LIN {X 0,Y 573.221,Z 156.08,A -85,B 0,C 180,E1 -2313.023,E2 -2313.023} C_VEL
LIN {X 0,Y 573.249,Z 156.083,A -85,B 0,C 180,E1 -2315.365,E2 -2315.365} C_VEL
LIN {X 0,Y 573.247,Z 156.077,A -85,B 0,C 180,E1 -2317.663,E2 -2317.663} C_VEL
LIN {X 0,Y 573.25,Z 156.08,A -85,B 0,C 180,E1 -2320.726,E2 -2320.726} C_VEL
LIN {X 0,Y 573.241,Z 156.081,A -85,B 0,C 180,E1 -2323.622,E2 -2323.622} C_VEL
LIN {X 0,Y 573.206,Z 156.082,A -85,B 0,C 180,E1 -2326.529,E2 -2326.529} C_VEL
LIN {X 0,Y 573.275,Z 156.074,A -85,B 0,C 180,E1 -2329.404,E2 -2329.404} C_VEL
LIN {X 0,Y 573.284,Z 156.078,A -85,B 0,C 180,E1 -2332.25,E2 -2332.25} C_VEL
LIN {X 0,Y 573.299,Z 156.071,A -85,B 0,C 180,E1 -2335.077,E2 -2335.077} C_VEL
LIN {X 0,Y 573.269,Z 156.075,A -85,B 0,C 180,E1 -2337.892,E2 -2337.892} C_VEL
LIN {X 0,Y 573.318,Z 156.074,A -85,B 0,C 180,E1 -2340.703,E2 -2340.703} C_VEL
LIN {X 0,Y 573.227,Z 156.079,A -85,B 0,C 180,E1 -2343.515,E2 -2343.515} C_VEL
LIN {X 0,Y 573.286,Z 156.077,A -85,B 0,C 180,E1 -2345.628,E2 -2345.628} C_VEL
LIN {X 0,Y 573.282,Z 156.073,A -85,B 0,C 180,E1 -2348.46,E2 -2348.46} C_VEL
LIN {X 0,Y 573.246,Z 156.078,A -85,B 0,C 180,E1 -2351.313,E2 -2351.313} C_VEL
LIN {X 0,Y 573.259,Z 156.078,A -85,B 0,C 180,E1 -2354.429,E2 -2354.429} C_VEL
LIN {X 0,Y 573.274,Z 156.074,A -85,B 0,C 180,E1 -2357.111,E2 -2357.111} C_VEL
LIN {X 0,Y 573.241,Z 156.077,A -85,B 0,C 180,E1 -2360.077,E2 -2360.077} C_VEL
LIN {X 0,Y 573.209,Z 156.082,A -85,B 0,C 180,E1 -2363.101,E2 -2363.101} C_VEL
LIN {X 0,Y 573.226,Z 156.08,A -85,B 0,C 180,E1 -2364.417,E2 -2364.417} C_VEL
LIN {X 0,Y 572.6,Z 156.16,A -85,B 0,C 180,E1 -2365.004,E2 -2365.004} C_VEL
LIN {X 0,Y 569.761,Z 156.517,A -85,B 0,C 180,E1 -2365.955,E2 -2365.955} C_VEL
LIN {X 0,Y 567.333,Z 156.82,A -85,B 0,C 180,E1 -2366.721,E2 -2366.721} C_VEL
LIN {X 0,Y 566.281,Z 156.947,A -85,B 0,C 180,E1 -2367.313,E2 -2367.313} C_VEL
LIN {X 0,Y 566.193,Z 156.957,A -85,B 0,C 180,E1 -2367.513,E2 -2367.513} C_VEL
LIN {X 0,Y 566.176,Z 156.959,A -85,B 0,C 180,E1 -2370.593,E2 -2370.593} C_VEL
LIN {X 0,Y 566.209,Z 156.955,A -85,B 0,C 180,E1 -2373.103,E2 -2373.103} C_VEL
LIN {X 0,Y 566.173,Z 156.961,A -85,B 0,C 180,E1 -2375.692,E2 -2375.692} C_VEL
LIN {X 0,Y 566.193,Z 156.955,A -85,B 0,C 180,E1 -2378.56,E2 -2378.56} C_VEL
LIN {X 0,Y 566.197,Z 156.96,A -85,B 0,C 180,E1 -2381.138,E2 -2381.138} C_VEL
LIN {X 0,Y 566.187,Z 156.958,A -85,B 0,C 180,E1 -2384.037,E2 -2384.037} C_VEL
LIN {X 0,Y 566.19,Z 156.956,A -85,B 0,C 180,E1 -2387.085,E2 -2387.085} C_VEL
LIN {X 0,Y 566.195,Z 156.958,A -85,B 0,C 180,E1 -2389.803,E2 -2389.803} C_VEL
LIN {X 0,Y 566.131,Z 156.967,A -85,B 0,C 180,E1 -2392.537,E2 -2392.537} C_VEL
LIN {X 0,Y 566.126,Z 159.575,A -85,B 0,C 180,E1 -2394.308,E2 -2394.308} C_VEL
LIN {X 0,Y 566.103,Z 163.804,A -85,B 0,C 180,E1 -2396.892,E2 -2396.892} C_VEL
LIN {X 0,Y 566.069,Z 167.996,A -85,B 0,C 180,E1 -2399.402,E2 -2399.402} C_VEL
LIN {X 0,Y 566.072,Z 172.14,A -85,B 0,C 180,E1 -2401.851,E2 -2401.851} C_VEL
LIN {X 0,Y 566.04,Z 177.644,A -85,B 0,C 180,E1 -2405.031,E2 -2405.031} C_VEL
LIN {X 0,Y 565.949,Z 181.747,A -85,B 0,C 180,E1 -2407.36,E2 -2407.36} C_VEL
LIN {X 0,Y 565.931,Z 187.178,A -85,B 0,C 180,E1 -2410.41,E2 -2410.41} C_VEL
LIN {X 0,Y 565.882,Z 192.758,A -85,B 0,C 180,E1 -2413.403,E2 -2413.403} C_VEL
LIN {X 0,Y 565.839,Z 196.558,A -85,B 0,C 180,E1 -2415.415,E2 -2415.415} C_VEL
LIN {X 0,Y 566.895,Z 204.229,A -85,B 0,C 180,E1 -2415.603,E2 -2415.603} C_VEL
LIN {X 0,Y 566.792,Z 217.644,A -85,B 0,C 180,E1 -2416.008,E2 -2416.008} C_VEL
LIN {X 0,Y 566.595,Z 230.276,A -85,B 0,C 180,E1 -2416.552,E2 -2416.552} C_VEL
LIN {X 0,Y 566.435,Z 241.516,A -85,B 0,C 180,E1 -2417.187,E2 -2417.187} C_VEL
LIN {X 0,Y 566.365,Z 252.951,A -85,B 0,C 180,E1 -2418.004,E2 -2418.004} C_VEL
LIN {X 0,Y 566.217,Z 262.307,A -85,B 0,C 180,E1 -2418.835,E2 -2418.835} C_VEL
LIN {X 0,Y 566.14,Z 271.26,A -85,B 0,C 180,E1 -2419.811,E2 -2419.811} C_VEL
LIN {X 0,Y 566.053,Z 279.323,A -85,B 0,C 180,E1 -2420.892,E2 -2420.892} C_VEL
LIN {X 0,Y 565.991,Z 284.78,A -85,B 0,C 180,E1 -2421.79,E2 -2421.79} C_VEL
LIN {X 0,Y 565.972,Z 290.113,A -85,B 0,C 180,E1 -2422.867,E2 -2422.867} C_VEL
LIN {X 0,Y 565.913,Z 294.264,A -85,B 0,C 180,E1 -2423.941,E2 -2423.941} C_VEL
LIN {X 0,Y 565.858,Z 297.355,A -85,B 0,C 180,E1 -2425.012,E2 -2425.012} C_VEL
LIN {X 0,Y 565.914,Z 298.89,A -85,B 0,C 180,E1 -2425.727,E2 -2425.727} C_VEL
LIN {X 0,Y 565.912,Z 299.981,A -85,B 0,C 180,E1 -2426.44,E2 -2426.44} C_VEL
LIN {X 0,Y 565.839,Z 300.967,A -85,B 0,C 180,E1 -2427.864,E2 -2427.864} C_VEL
LIN {X 0,Y 565.845,Z 300.887,A -85,B 0,C 180,E1 -2428.576,E2 -2428.576} C_VEL
LIN {X 0,Y 565.841,Z 300.384,A -85,B 0,C 180,E1 -2429.288,E2 -2429.288} C_VEL
LIN {X 0,Y 565.843,Z 298.185,A -85,B 0,C 180,E1 -2430.711,E2 -2430.711} C_VEL
LIN {X 0,Y 565.908,Z 295.441,A -85,B 0,C 180,E1 -2431.779,E2 -2431.779} C_VEL
LIN {X 0,Y 565.902,Z 291.689,A -85,B 0,C 180,E1 -2432.847,E2 -2432.847} C_VEL
LIN {X 0,Y 566.003,Z 286.823,A -85,B 0,C 180,E1 -2433.915,E2 -2433.915} C_VEL
LIN {X 0,Y 566.047,Z 280.702,A -85,B 0,C 180,E1 -2434.985,E2 -2434.985} C_VEL
LIN {X 0,Y 566.111,Z 273.096,A -85,B 0,C 180,E1 -2436.056,E2 -2436.056} C_VEL
LIN {X 0,Y 566.191,Z 265.345,A -85,B 0,C 180,E1 -2436.948,E2 -2436.948} C_VEL
LIN {X 0,Y 566.321,Z 254.772,A -85,B 0,C 180,E1 -2437.935,E2 -2437.935} C_VEL
LIN {X 0,Y 566.454,Z 244.034,A -85,B 0,C 180,E1 -2438.741,E2 -2438.741} C_VEL
LIN {X 0,Y 566.563,Z 233.576,A -85,B 0,C 180,E1 -2439.369,E2 -2439.369} C_VEL
LIN {X 0,Y 566.742,Z 221.019,A -85,B 0,C 180,E1 -2439.951,E2 -2439.951} C_VEL
LIN {X 0,Y 566.873,Z 207.708,A -85,B 0,C 180,E1 -2440.4,E2 -2440.4} C_VEL
LIN {X 0,Y 566.719,Z 201.824,A -85,B 0,C 180,E1 -2440.55,E2 -2440.55} C_VEL
LIN {X 0,Y 565.896,Z 196.528,A -85,B 0,C 180,E1 -2440.69,E2 -2440.69} C_VEL
LIN {X 0,Y 565.922,Z 190.956,A -85,B 0,C 180,E1 -2443.646,E2 -2443.646} C_VEL
LIN {X 0,Y 565.91,Z 186.866,A -85,B 0,C 180,E1 -2445.854,E2 -2445.854} C_VEL
LIN {X 0,Y 565.974,Z 182.892,A -85,B 0,C 180,E1 -2448.084,E2 -2448.084} C_VEL
LIN {X 0,Y 566.027,Z 177.535,A -85,B 0,C 180,E1 -2451.103,E2 -2451.103} C_VEL
LIN {X 0,Y 566.052,Z 172.237,A -85,B 0,C 180,E1 -2454.185,E2 -2454.185} C_VEL
LIN {X 0,Y 566.089,Z 166.881,A -85,B 0,C 180,E1 -2457.343,E2 -2457.343} C_VEL
LIN {X 0,Y 566.106,Z 162.848,A -85,B 0,C 180,E1 -2459.771,E2 -2459.771} C_VEL
LIN {X 0,Y 566.117,Z 158.483,A -85,B 0,C 180,E1 -2462.415,E2 -2462.415} C_VEL
LIN {X 0,Y 566.1,Z 157.355,A -85,B 0,C 180,E1 -2463.107,E2 -2463.107} C_VEL
LIN {X 0,Y 566.162,Z 156.96,A -85,B 0,C 180,E1 -2463.956,E2 -2463.956} C_VEL
LIN {X 0,Y 566.168,Z 156.963,A -85,B 0,C 180,E1 -2466.569,E2 -2466.569} C_VEL
LIN {X 0,Y 566.199,Z 156.954,A -85,B 0,C 180,E1 -2469.271,E2 -2469.271} C_VEL
LIN {X 0,Y 566.209,Z 156.958,A -85,B 0,C 180,E1 -2472.083,E2 -2472.083} C_VEL
LIN {X 0,Y 566.154,Z 156.961,A -85,B 0,C 180,E1 -2475.033,E2 -2475.033} C_VEL
LIN {X 0,Y 566.209,Z 156.952,A -85,B 0,C 180,E1 -2478.132,E2 -2478.132} C_VEL
LIN {X 0,Y 566.199,Z 156.961,A -85,B 0,C 180,E1 -2480.725,E2 -2480.725} C_VEL
LIN {X 0,Y 566.175,Z 156.96,A -85,B 0,C 180,E1 -2483.783,E2 -2483.783} C_VEL
LIN {X 0,Y 566.202,Z 156.954,A -85,B 0,C 180,E1 -2486.896,E2 -2486.896} C_VEL
LIN {X 0,Y 566.17,Z 156.964,A -85,B 0,C 180,E1 -2489.406,E2 -2489.406} C_VEL
LIN {X 0,Y 566.196,Z 156.954,A -85,B 0,C 180,E1 -2491.856,E2 -2491.856} C_VEL
LIN {X 0,Y 566.202,Z 156.956,A -85,B 0,C 180,E1 -2494.25,E2 -2494.25} C_VEL
LIN {X 0,Y 566.22,Z 156.954,A -85,B 0,C 180,E1 -2496.697,E2 -2496.697} C_VEL
LIN {X 0,Y 566.184,Z 156.96,A -85,B 0,C 180,E1 -2499.661,E2 -2499.661} C_VEL
LIN {X 0,Y 566.214,Z 156.954,A -85,B 0,C 180,E1 -2502.875,E2 -2502.875} C_VEL
LIN {X 0,Y 566.205,Z 156.955,A -85,B 0,C 180,E1 -2505.626,E2 -2505.626} C_VEL
LIN {X 0,Y 566.254,Z 156.953,A -85,B 0,C 180,E1 -2508.643,E2 -2508.643} C_VEL
LIN {X 0,Y 566.226,Z 156.951,A -85,B 0,C 180,E1 -2511.434,E2 -2511.434} C_VEL
LIN {X 0,Y 566.212,Z 156.956,A -85,B 0,C 180,E1 -2513.586,E2 -2513.586} C_VEL
LIN {X 0,Y 566.165,Z 156.963,A -85,B 0,C 180,E1 -2515.728,E2 -2515.728} C_VEL
LIN {X 0,Y 566.236,Z 156.951,A -85,B 0,C 180,E1 -2517.866,E2 -2517.866} C_VEL
LIN {X 0,Y 566.278,Z 156.95,A -85,B 0,C 180,E1 -2520.711,E2 -2520.711} C_VEL
LIN {X 0,Y 566.17,Z 156.958,A -85,B 0,C 180,E1 -2523.558,E2 -2523.558} C_VEL
LIN {X 0,Y 566.25,Z 156.951,A -85,B 0,C 180,E1 -2525.698,E2 -2525.698} C_VEL
LIN {X 0,Y 566.229,Z 156.956,A -85,B 0,C 180,E1 -2527.847,E2 -2527.847} C_VEL
LIN {X 0,Y 566.245,Z 156.949,A -85,B 0,C 180,E1 -2530.729,E2 -2530.729} C_VEL
LIN {X 0,Y 566.18,Z 156.957,A -85,B 0,C 180,E1 -2533.641,E2 -2533.641} C_VEL
LIN {X 0,Y 566.188,Z 156.962,A -85,B 0,C 180,E1 -2536.588,E2 -2536.588} C_VEL
LIN {X 0,Y 566.179,Z 156.959,A -85,B 0,C 180,E1 -2539.582,E2 -2539.582} C_VEL
LIN {X 0,Y 566.193,Z 156.955,A -85,B 0,C 180,E1 -2542.631,E2 -2542.631} C_VEL
LIN {X 0,Y 566.215,Z 156.957,A -85,B 0,C 180,E1 -2545.039,E2 -2545.039} C_VEL
LIN {X 0,Y 566.199,Z 156.956,A -85,B 0,C 180,E1 -2547.34,E2 -2547.34} C_VEL
LIN {X 0,Y 566.201,Z 156.954,A -85,B 0,C 180,E1 -2549.769,E2 -2549.769} C_VEL
LIN {X 0,Y 566.177,Z 156.961,A -85,B 0,C 180,E1 -2552.433,E2 -2552.433} C_VEL
LIN {X 0,Y 566.171,Z 156.958,A -85,B 0,C 180,E1 -2554.995,E2 -2554.995} C_VEL
LIN {X 0,Y 566.17,Z 156.964,A -85,B 0,C 180,E1 -2557.463,E2 -2557.463} C_VEL
LIN {X 0,Y 566.203,Z 156.954,A -85,B 0,C 180,E1 -2560.2,E2 -2560.2} C_VEL
LIN {X 0,Y 566.19,Z 156.957,A -85,B 0,C 180,E1 -2563.055,E2 -2563.055} C_VEL
LIN {X 0,Y 566.182,Z 156.963,A -85,B 0,C 180,E1 -2566.051,E2 -2566.051} C_VEL
LIN {X 0,Y 566.193,Z 156.956,A -85,B 0,C 180,E1 -2568.866,E2 -2568.866} C_VEL
LIN {X 0,Y 566.162,Z 156.964,A -85,B 0,C 180,E1 -2571.639,E2 -2571.639} C_VEL
LIN {X 0,Y 566.212,Z 157.121,A -85,B 0,C 180,E1 -2573.64,E2 -2573.64} C_VEL
LIN {X 0,Y 566.507,Z 161.011,A -85,B 0,C 180,E1 -2575.207,E2 -2575.207} C_VEL
LIN {X 0,Y 566.419,Z 167.636,A -85,B 0,C 180,E1 -2577.759,E2 -2577.759} C_VEL
LIN {X 0,Y 566.362,Z 174.512,A -85,B 0,C 180,E1 -2580.3,E2 -2580.3} C_VEL
LIN {X 0,Y 566.272,Z 181.071,A -85,B 0,C 180,E1 -2582.667,E2 -2582.667} C_VEL
LIN {X 0,Y 566.22,Z 188.951,A -85,B 0,C 180,E1 -2585.432,E2 -2585.432} C_VEL
LIN {X 0,Y 566.161,Z 198.194,A -85,B 0,C 180,E1 -2588.593,E2 -2588.593} C_VEL
LIN {X 0,Y 566.073,Z 207.033,A -85,B 0,C 180,E1 -2591.545,E2 -2591.545} C_VEL
LIN {X 0,Y 566.02,Z 215.94,A -85,B 0,C 180,E1 -2594.518,E2 -2594.518} C_VEL
LIN {X 0,Y 565.949,Z 223.731,A -85,B 0,C 180,E1 -2597.085,E2 -2597.085} C_VEL
LIN {X 0,Y 565.948,Z 224.496,A -85,B 0,C 180,E1 -2597.336,E2 -2597.336} C_VEL
LIN {X 0,Y 566.94,Z 231.578,A -85,B 0,C 180,E1 -2597.495,E2 -2597.495} C_VEL
LIN {X 0,Y 566.82,Z 243.914,A -85,B 0,C 180,E1 -2597.833,E2 -2597.833} C_VEL
LIN {X 0,Y 566.641,Z 256.933,A -85,B 0,C 180,E1 -2598.347,E2 -2598.347} C_VEL
LIN {X 0,Y 566.524,Z 268.514,A -85,B 0,C 180,E1 -2598.956,E2 -2598.956} C_VEL
LIN {X 0,Y 566.43,Z 279.938,A -85,B 0,C 180,E1 -2599.727,E2 -2599.727} C_VEL
LIN {X 0,Y 566.281,Z 289.613,A -85,B 0,C 180,E1 -2600.536,E2 -2600.536} C_VEL
LIN {X 0,Y 566.18,Z 298.423,A -85,B 0,C 180,E1 -2601.435,E2 -2601.435} C_VEL
LIN {X 0,Y 566.055,Z 307.009,A -85,B 0,C 180,E1 -2602.51,E2 -2602.51} C_VEL
LIN {X 0,Y 565.964,Z 313.874,A -85,B 0,C 180,E1 -2603.584,E2 -2603.584} C_VEL
LIN {X 0,Y 565.937,Z 319.37,A -85,B 0,C 180,E1 -2604.657,E2 -2604.657} C_VEL
LIN {X 0,Y 565.959,Z 323.68,A -85,B 0,C 180,E1 -2605.728,E2 -2605.728} C_VEL
LIN {X 0,Y 565.927,Z 325.96,A -85,B 0,C 180,E1 -2606.441,E2 -2606.441} C_VEL
LIN {X 0,Y 565.878,Z 327.809,A -85,B 0,C 180,E1 -2607.153,E2 -2607.153} C_VEL
LIN {X 0,Y 565.846,Z 330.185,A -85,B 0,C 180,E1 -2608.577,E2 -2608.577} C_VEL
LIN {X 0,Y 565.839,Z 331,A -85,B 0,C 180,E1 -2610,E2 -2610} C_VEL
LIN {X 0,Y 565.846,Z 330.185,A -85,B 0,C 180,E1 -2611.424,E2 -2611.424} C_VEL
LIN {X 0,Y 565.878,Z 327.809,A -85,B 0,C 180,E1 -2612.848,E2 -2612.848} C_VEL
LIN {X 0,Y 565.926,Z 324.895,A -85,B 0,C 180,E1 -2613.917,E2 -2613.917} C_VEL
LIN {X 0,Y 565.878,Z 320.948,A -85,B 0,C 180,E1 -2614.988,E2 -2614.988} C_VEL
LIN {X 0,Y 566.002,Z 315.867,A -85,B 0,C 180,E1 -2616.059,E2 -2616.059} C_VEL
LIN {X 0,Y 566.04,Z 309.468,A -85,B 0,C 180,E1 -2617.132,E2 -2617.132} C_VEL
LIN {X 0,Y 566.133,Z 301.479,A -85,B 0,C 180,E1 -2618.208,E2 -2618.208} C_VEL
LIN {X 0,Y 566.229,Z 293.336,A -85,B 0,C 180,E1 -2619.105,E2 -2619.105} C_VEL
LIN {X 0,Y 566.335,Z 283.402,A -85,B 0,C 180,E1 -2620.005,E2 -2620.005} C_VEL
LIN {X 0,Y 566.467,Z 272.339,A -85,B 0,C 180,E1 -2620.805,E2 -2620.805} C_VEL
LIN {X 0,Y 566.607,Z 259.952,A -85,B 0,C 180,E1 -2621.51,E2 -2621.51} C_VEL
LIN {X 0,Y 566.753,Z 247.779,A -85,B 0,C 180,E1 -2622.033,E2 -2622.033} C_VEL
LIN {X 0,Y 566.903,Z 234.363,A -85,B 0,C 180,E1 -2622.439,E2 -2622.439} C_VEL
LIN {X 0,Y 566.629,Z 228.833,A -85,B 0,C 180,E1 -2622.567,E2 -2622.567} C_VEL
LIN {X 0,Y 565.947,Z 224.493,A -85,B 0,C 180,E1 -2622.665,E2 -2622.665} C_VEL
LIN {X 0,Y 566.017,Z 217.05,A -85,B 0,C 180,E1 -2625.114,E2 -2625.114} C_VEL
LIN {X 0,Y 566.057,Z 208.146,A -85,B 0,C 180,E1 -2628.082,E2 -2628.082} C_VEL
LIN {X 0,Y 566.101,Z 200.223,A -85,B 0,C 180,E1 -2630.72,E2 -2630.72} C_VEL
LIN {X 0,Y 566.172,Z 192.343,A -85,B 0,C 180,E1 -2633.403,E2 -2633.403} C_VEL
LIN {X 0,Y 566.247,Z 184.417,A -85,B 0,C 180,E1 -2636.141,E2 -2636.141} C_VEL
LIN {X 0,Y 566.339,Z 176.561,A -85,B 0,C 180,E1 -2638.943,E2 -2638.943} C_VEL
LIN {X 0,Y 566.4,Z 169.86,A -85,B 0,C 180,E1 -2641.407,E2 -2641.407} C_VEL
LIN {X 0,Y 566.475,Z 163.253,A -85,B 0,C 180,E1 -2643.936,E2 -2643.936} C_VEL
LIN {X 0,Y 566.491,Z 158.911,A -85,B 0,C 180,E1 -2645.666,E2 -2645.666} C_VEL
LIN {X 0,Y 566.195,Z 156.962,A -85,B 0,C 180,E1 -2646.568,E2 -2646.568} C_VEL
LIN {X 0,Y 566.193,Z 156.959,A -85,B 0,C 180,E1 -2649.683,E2 -2649.683} C_VEL
LIN {X 0,Y 566.213,Z 156.957,A -85,B 0,C 180,E1 -2652.084,E2 -2652.084} C_VEL
LIN {X 0,Y 566.158,Z 156.963,A -85,B 0,C 180,E1 -2655.034,E2 -2655.034} C_VEL
LIN {X 0,Y 566.174,Z 156.958,A -85,B 0,C 180,E1 -2657.909,E2 -2657.909} C_VEL
LIN {X 0,Y 566.199,Z 156.956,A -85,B 0,C 180,E1 -2660.725,E2 -2660.725} C_VEL
LIN {X 0,Y 566.198,Z 156.959,A -85,B 0,C 180,E1 -2663.782,E2 -2663.782} C_VEL
LIN {X 0,Y 566.208,Z 156.953,A -85,B 0,C 180,E1 -2666.261,E2 -2666.261} C_VEL
LIN {X 0,Y 566.182,Z 156.961,A -85,B 0,C 180,E1 -2668.919,E2 -2668.919} C_VEL
LIN {X 0,Y 566.17,Z 156.959,A -85,B 0,C 180,E1 -2671.045,E2 -2671.045} C_VEL
LIN {X 0,Y 566.186,Z 156.959,A -85,B 0,C 180,E1 -2673.457,E2 -2673.457} C_VEL
LIN {X 0,Y 566.191,Z 156.957,A -85,B 0,C 180,E1 -2675.819,E2 -2675.819} C_VEL
LIN {X 0,Y 566.19,Z 156.959,A -85,B 0,C 180,E1 -2678.576,E2 -2678.576} C_VEL
LIN {X 0,Y 566.194,Z 156.955,A -85,B 0,C 180,E1 -2681.172,E2 -2681.172} C_VEL
LIN {X 0,Y 566.207,Z 156.955,A -85,B 0,C 180,E1 -2683.412,E2 -2683.412} C_VEL
LIN {X 0,Y 566.168,Z 156.959,A -85,B 0,C 180,E1 -2686.358,E2 -2686.358} C_VEL
LIN {X 0,Y 566.25,Z 156.95,A -85,B 0,C 180,E1 -2689.271,E2 -2689.271} C_VEL
LIN {X 0,Y 566.235,Z 156.955,A -85,B 0,C 180,E1 -2692.153,E2 -2692.153} C_VEL
LIN {X 0,Y 566.27,Z 156.946,A -85,B 0,C 180,E1 -2695.016,E2 -2695.016} C_VEL
LIN {X 0,Y 566.241,Z 156.95,A -85,B 0,C 180,E1 -2697.866,E2 -2697.866} C_VEL
LIN {X 0,Y 566.286,Z 156.949,A -85,B 0,C 180,E1 -2700.711,E2 -2700.711} C_VEL
LIN {X 0,Y 566.179,Z 156.958,A -85,B 0,C 180,E1 -2703.559,E2 -2703.559} C_VEL
LIN {X 0,Y 566.253,Z 156.954,A -85,B 0,C 180,E1 -2705.699,E2 -2705.699} C_VEL
LIN {X 0,Y 566.224,Z 156.953,A -85,B 0,C 180,E1 -2708.566,E2 -2708.566} C_VEL
LIN {X 0,Y 566.212,Z 156.953,A -85,B 0,C 180,E1 -2711.455,E2 -2711.455} C_VEL
LIN {X 0,Y 566.211,Z 156.955,A -85,B 0,C 180,E1 -2714.511,E2 -2714.511} C_VEL
LIN {X 0,Y 566.23,Z 156.954,A -85,B 0,C 180,E1 -2717.331,E2 -2717.331} C_VEL
LIN {X 0,Y 566.202,Z 156.955,A -85,B 0,C 180,E1 -2720.338,E2 -2720.338} C_VEL
LIN {X 0,Y 566.166,Z 156.959,A -85,B 0,C 180,E1 -2723.405,E2 -2723.405} C_VEL
LIN {X 0,Y 566.199,Z 156.96,A -85,B 0,C 180,E1 -2725.75,E2 -2725.75} C_VEL
LIN {X 0,Y 566.193,Z 156.957,A -85,B 0,C 180,E1 -2727.513,E2 -2727.513} C_VEL
LIN {X 0,Y 565.516,Z 157.041,A -85,B 0,C 180,E1 -2728.107,E2 -2728.107} C_VEL
LIN {X 0,Y 562.651,Z 157.4,A -85,B 0,C 180,E1 -2729.071,E2 -2729.071} C_VEL
LIN {X 0,Y 560.241,Z 157.697,A -85,B 0,C 180,E1 -2729.846,E2 -2729.846} C_VEL
LIN {X 0,Y 559.214,Z 157.825,A -85,B 0,C 180,E1 -2730.445,E2 -2730.445} C_VEL
LIN {X 0,Y 559.134,Z 157.836,A -85,B 0,C 180,E1 -2730.648,E2 -2730.648} C_VEL
LIN {X 0,Y 559.156,Z 157.832,A -85,B 0,C 180,E1 -2733.576,E2 -2733.576} C_VEL
LIN {X 0,Y 559.138,Z 157.836,A -85,B 0,C 180,E1 -2736.449,E2 -2736.449} C_VEL
LIN {X 0,Y 559.158,Z 157.833,A -85,B 0,C 180,E1 -2738.936,E2 -2738.936} C_VEL
LIN {X 0,Y 559.177,Z 157.829,A -85,B 0,C 180,E1 -2741.77,E2 -2741.77} C_VEL
LIN {X 0,Y 559.127,Z 157.838,A -85,B 0,C 180,E1 -2744.741,E2 -2744.741} C_VEL
LIN {X 0,Y 559.162,Z 157.837,A -85,B 0,C 180,E1 -2747.865,E2 -2747.865} C_VEL
LIN {X 0,Y 559.16,Z 157.838,A -85,B 0,C 180,E1 -2751.067,E2 -2751.067} C_VEL
LIN {X 0,Y 559.082,Z 157.843,A -85,B 0,C 180,E1 -2752.369,E2 -2752.369} C_VEL
LIN {X 0,Y 559.067,Z 158.162,A -85,B 0,C 180,E1 -2752.888,E2 -2752.888} C_VEL
LIN {X 0,Y 559.057,Z 162.433,A -85,B 0,C 180,E1 -2755.551,E2 -2755.551} C_VEL
LIN {X 0,Y 559.063,Z 167.634,A -85,B 0,C 180,E1 -2758.742,E2 -2758.742} C_VEL
LIN {X 0,Y 559.028,Z 172.498,A -85,B 0,C 180,E1 -2761.647,E2 -2761.647} C_VEL
LIN {X 0,Y 558.969,Z 177.982,A -85,B 0,C 180,E1 -2764.86,E2 -2764.86} C_VEL
LIN {X 0,Y 558.869,Z 183.196,A -85,B 0,C 180,E1 -2767.837,E2 -2767.837} C_VEL
LIN {X 0,Y 558.839,Z 188.631,A -85,B 0,C 180,E1 -2770.915,E2 -2770.915} C_VEL
LIN {X 0,Y 558.815,Z 192.708,A -85,B 0,C 180,E1 -2773.187,E2 -2773.187} C_VEL
LIN {X 0,Y 558.744,Z 196.529,A -85,B 0,C 180,E1 -2775.236,E2 -2775.236} C_VEL
LIN {X 0,Y 559.952,Z 204.885,A -85,B 0,C 180,E1 -2775.463,E2 -2775.463} C_VEL
LIN {X 0,Y 559.839,Z 218.126,A -85,B 0,C 180,E1 -2775.874,E2 -2775.874} C_VEL
LIN {X 0,Y 559.656,Z 229.785,A -85,B 0,C 180,E1 -2776.382,E2 -2776.382} C_VEL
LIN {X 0,Y 559.443,Z 241.118,A -85,B 0,C 180,E1 -2777.024,E2 -2777.024} C_VEL
LIN {X 0,Y 559.354,Z 252.632,A -85,B 0,C 180,E1 -2777.851,E2 -2777.851} C_VEL
LIN {X 0,Y 559.18,Z 262.807,A -85,B 0,C 180,E1 -2778.77,E2 -2778.77} C_VEL
LIN {X 0,Y 559.099,Z 272.547,A -85,B 0,C 180,E1 -2779.864,E2 -2779.864} C_VEL
LIN {X 0,Y 558.978,Z 280.34,A -85,B 0,C 180,E1 -2780.958,E2 -2780.958} C_VEL
LIN {X 0,Y 558.895,Z 286.57,A -85,B 0,C 180,E1 -2782.049,E2 -2782.049} C_VEL
LIN {X 0,Y 558.887,Z 291.516,A -85,B 0,C 180,E1 -2783.139,E2 -2783.139} C_VEL
LIN {X 0,Y 558.847,Z 295.329,A -85,B 0,C 180,E1 -2784.226,E2 -2784.226} C_VEL
LIN {X 0,Y 558.775,Z 297.293,A -85,B 0,C 180,E1 -2784.949,E2 -2784.949} C_VEL
LIN {X 0,Y 558.808,Z 298.841,A -85,B 0,C 180,E1 -2785.672,E2 -2785.672} C_VEL
LIN {X 0,Y 558.821,Z 299.953,A -85,B 0,C 180,E1 -2786.395,E2 -2786.395} C_VEL
LIN {X 0,Y 558.745,Z 300.961,A -85,B 0,C 180,E1 -2787.837,E2 -2787.837} C_VEL
LIN {X 0,Y 558.744,Z 300.893,A -85,B 0,C 180,E1 -2788.558,E2 -2788.558} C_VEL
LIN {X 0,Y 558.741,Z 300.411,A -85,B 0,C 180,E1 -2789.279,E2 -2789.279} C_VEL
LIN {X 0,Y 558.744,Z 298.234,A -85,B 0,C 180,E1 -2790.72,E2 -2790.72} C_VEL
LIN {X 0,Y 558.824,Z 295.514,A -85,B 0,C 180,E1 -2791.801,E2 -2791.801} C_VEL
LIN {X 0,Y 558.826,Z 291.787,A -85,B 0,C 180,E1 -2792.883,E2 -2792.883} C_VEL
LIN {X 0,Y 558.908,Z 286.948,A -85,B 0,C 180,E1 -2793.965,E2 -2793.965} C_VEL
LIN {X 0,Y 558.972,Z 280.856,A -85,B 0,C 180,E1 -2795.048,E2 -2795.048} C_VEL
LIN {X 0,Y 559.07,Z 273.29,A -85,B 0,C 180,E1 -2796.133,E2 -2796.133} C_VEL
LIN {X 0,Y 559.181,Z 263.792,A -85,B 0,C 180,E1 -2797.219,E2 -2797.219} C_VEL
LIN {X 0,Y 559.368,Z 253.999,A -85,B 0,C 180,E1 -2798.125,E2 -2798.125} C_VEL
LIN {X 0,Y 559.48,Z 243.037,A -85,B 0,C 180,E1 -2798.942,E2 -2798.942} C_VEL
LIN {X 0,Y 559.646,Z 232.311,A -85,B 0,C 180,E1 -2799.577,E2 -2799.577} C_VEL
LIN {X 0,Y 559.812,Z 220.513,A -85,B 0,C 180,E1 -2800.122,E2 -2800.122} C_VEL
LIN {X 0,Y 559.937,Z 207.79,A -85,B 0,C 180,E1 -2800.553,E2 -2800.553} C_VEL
LIN {X 0,Y 559.828,Z 202.867,A -85,B 0,C 180,E1 -2800.681,E2 -2800.681} C_VEL
LIN {X 0,Y 558.815,Z 196.534,A -85,B 0,C 180,E1 -2800.85,E2 -2800.85} C_VEL
LIN {X 0,Y 558.834,Z 191.043,A -85,B 0,C 180,E1 -2803.823,E2 -2803.823} C_VEL
LIN {X 0,Y 558.872,Z 185.73,A -85,B 0,C 180,E1 -2806.81,E2 -2806.81} C_VEL
LIN {X 0,Y 558.91,Z 181.128,A -85,B 0,C 180,E1 -2809.422,E2 -2809.422} C_VEL
LIN {X 0,Y 558.952,Z 176.384,A -85,B 0,C 180,E1 -2812.159,E2 -2812.159} C_VEL
LIN {X 0,Y 559.012,Z 171.305,A -85,B 0,C 180,E1 -2815.149,E2 -2815.149} C_VEL
LIN {X 0,Y 559.026,Z 167.019,A -85,B 0,C 180,E1 -2817.718,E2 -2817.718} C_VEL
LIN {X 0,Y 559.121,Z 161.593,A -85,B 0,C 180,E1 -2821.018,E2 -2821.018} C_VEL
LIN {X 0,Y 559.05,Z 158.835,A -85,B 0,C 180,E1 -2822.719,E2 -2822.719} C_VEL
LIN {X 0,Y 559.072,Z 157.846,A -85,B 0,C 180,E1 -2823.578,E2 -2823.578} C_VEL
LIN {X 0,Y 559.115,Z 157.84,A -85,B 0,C 180,E1 -2826.44,E2 -2826.44} C_VEL
LIN {X 0,Y 559.158,Z 157.833,A -85,B 0,C 180,E1 -2828.931,E2 -2828.931} C_VEL
LIN {X 0,Y 559.18,Z 157.833,A -85,B 0,C 180,E1 -2831.764,E2 -2831.764} C_VEL
LIN {X 0,Y 559.121,Z 157.836,A -85,B 0,C 180,E1 -2834.736,E2 -2834.736} C_VEL
LIN {X 0,Y 559.152,Z 157.838,A -85,B 0,C 180,E1 -2837.255,E2 -2837.255} C_VEL
LIN {X 0,Y 559.163,Z 157.831,A -85,B 0,C 180,E1 -2840.132,E2 -2840.132} C_VEL
LIN {X 0,Y 559.117,Z 157.838,A -85,B 0,C 180,E1 -2842.889,E2 -2842.889} C_VEL
LIN {X 0,Y 559.147,Z 157.839,A -85,B 0,C 180,E1 -2846.047,E2 -2846.047} C_VEL
LIN {X 0,Y 559.141,Z 157.836,A -85,B 0,C 180,E1 -2848.979,E2 -2848.979} C_VEL
LIN {X 0,Y 559.165,Z 157.832,A -85,B 0,C 180,E1 -2851.611,E2 -2851.611} C_VEL
LIN {X 0,Y 559.175,Z 157.829,A -85,B 0,C 180,E1 -2853.902,E2 -2853.902} C_VEL
LIN {X 0,Y 559.15,Z 157.832,A -85,B 0,C 180,E1 -2857.067,E2 -2857.067} C_VEL
LIN {X 0,Y 559.151,Z 157.834,A -85,B 0,C 180,E1 -2859.394,E2 -2859.394} C_VEL
LIN {X 0,Y 559.137,Z 157.834,A -85,B 0,C 180,E1 -2862.442,E2 -2862.442} C_VEL
LIN {X 0,Y 559.156,Z 157.835,A -85,B 0,C 180,E1 -2865.441,E2 -2865.441} C_VEL
LIN {X 0,Y 559.237,Z 157.828,A -85,B 0,C 180,E1 -2868.566,E2 -2868.566} C_VEL
LIN {X 0,Y 559.179,Z 157.828,A -85,B 0,C 180,E1 -2871.325,E2 -2871.325} C_VEL
LIN {X 0,Y 559.175,Z 157.831,A -85,B 0,C 180,E1 -2873.505,E2 -2873.505} C_VEL
LIN {X 0,Y 559.124,Z 157.841,A -85,B 0,C 180,E1 -2875.675,E2 -2875.675} C_VEL
LIN {X 0,Y 559.208,Z 157.826,A -85,B 0,C 180,E1 -2877.839,E2 -2877.839} C_VEL
LIN {X 0,Y 559.246,Z 157.826,A -85,B 0,C 180,E1 -2880.72,E2 -2880.72} C_VEL
LIN {X 0,Y 559.221,Z 157.826,A -85,B 0,C 180,E1 -2882.881,E2 -2882.881} C_VEL
LIN {X 0,Y 559.219,Z 157.828,A -85,B 0,C 180,E1 -2885.77,E2 -2885.77} C_VEL
LIN {X 0,Y 559.192,Z 157.831,A -85,B 0,C 180,E1 -2887.946,E2 -2887.946} C_VEL
LIN {X 0,Y 559.223,Z 157.825,A -85,B 0,C 180,E1 -2890.866,E2 -2890.866} C_VEL
LIN {X 0,Y 559.15,Z 157.832,A -85,B 0,C 180,E1 -2893.816,E2 -2893.816} C_VEL
LIN {X 0,Y 559.151,Z 157.836,A -85,B 0,C 180,E1 -2896.803,E2 -2896.803} C_VEL
LIN {X 0,Y 559.14,Z 157.839,A -85,B 0,C 180,E1 -2899.839,E2 -2899.839} C_VEL
LIN {X 0,Y 559.132,Z 157.836,A -85,B 0,C 180,E1 -2902.153,E2 -2902.153} C_VEL
LIN {X 0,Y 559.149,Z 157.832,A -85,B 0,C 180,E1 -2904.505,E2 -2904.505} C_VEL
LIN {X 0,Y 559.165,Z 157.837,A -85,B 0,C 180,E1 -2906.903,E2 -2906.903} C_VEL
LIN {X 0,Y 559.162,Z 157.831,A -85,B 0,C 180,E1 -2909.868,E2 -2909.868} C_VEL
LIN {X 0,Y 559.145,Z 157.834,A -85,B 0,C 180,E1 -2912.716,E2 -2912.716} C_VEL
LIN {X 0,Y 559.118,Z 157.839,A -85,B 0,C 180,E1 -2915.325,E2 -2915.325} C_VEL
LIN {X 0,Y 559.11,Z 157.838,A -85,B 0,C 180,E1 -2918.019,E2 -2918.019} C_VEL
LIN {X 0,Y 559.156,Z 157.838,A -85,B 0,C 180,E1 -2920.813,E2 -2920.813} C_VEL
LIN {X 0,Y 559.142,Z 157.833,A -85,B 0,C 180,E1 -2923.734,E2 -2923.734} C_VEL
LIN {X 0,Y 559.153,Z 157.833,A -85,B 0,C 180,E1 -2926.803,E2 -2926.803} C_VEL
LIN {X 0,Y 559.158,Z 157.835,A -85,B 0,C 180,E1 -2929.192,E2 -2929.192} C_VEL
LIN {X 0,Y 559.112,Z 157.84,A -85,B 0,C 180,E1 -2931.985,E2 -2931.985} C_VEL
LIN {X 0,Y 559.182,Z 157.867,A -85,B 0,C 180,E1 -2933.44,E2 -2933.44} C_VEL
LIN {X 0,Y 559.511,Z 162.058,A -85,B 0,C 180,E1 -2935.156,E2 -2935.156} C_VEL
LIN {X 0,Y 559.403,Z 168.682,A -85,B 0,C 180,E1 -2937.737,E2 -2937.737} C_VEL
LIN {X 0,Y 559.357,Z 176.502,A -85,B 0,C 180,E1 -2940.662,E2 -2940.662} C_VEL
LIN {X 0,Y 559.226,Z 185.472,A -85,B 0,C 180,E1 -2943.908,E2 -2943.908} C_VEL
LIN {X 0,Y 559.138,Z 193.056,A -85,B 0,C 180,E1 -2946.573,E2 -2946.573} C_VEL
LIN {X 0,Y 559.04,Z 201.23,A -85,B 0,C 180,E1 -2949.392,E2 -2949.392} C_VEL
LIN {X 0,Y 559.002,Z 209.142,A -85,B 0,C 180,E1 -2952.062,E2 -2952.062} C_VEL
LIN {X 0,Y 558.938,Z 217.053,A -85,B 0,C 180,E1 -2954.691,E2 -2954.691} C_VEL
LIN {X 0,Y 558.886,Z 224.496,A -85,B 0,C 180,E1 -2957.173,E2 -2957.173} C_VEL
LIN {X 0,Y 559.994,Z 232.577,A -85,B 0,C 180,E1 -2957.36,E2 -2957.36} C_VEL
LIN {X 0,Y 559.859,Z 245.344,A -85,B 0,C 180,E1 -2957.73,E2 -2957.73} C_VEL
LIN {X 0,Y 559.686,Z 258.27,A -85,B 0,C 180,E1 -2958.262,E2 -2958.262} C_VEL
LIN {X 0,Y 559.536,Z 268.976,A -85,B 0,C 180,E1 -2958.844,E2 -2958.844} C_VEL
LIN {X 0,Y 559.418,Z 279.937,A -85,B 0,C 180,E1 -2959.597,E2 -2959.597} C_VEL
LIN {X 0,Y 559.242,Z 289.612,A -85,B 0,C 180,E1 -2960.416,E2 -2960.416} C_VEL
LIN {X 0,Y 559.126,Z 298.423,A -85,B 0,C 180,E1 -2961.326,E2 -2961.326} C_VEL
LIN {X 0,Y 558.995,Z 307.01,A -85,B 0,C 180,E1 -2962.415,E2 -2962.415} C_VEL
LIN {X 0,Y 558.884,Z 314.691,A -85,B 0,C 180,E1 -2963.65,E2 -2963.65} C_VEL
LIN {X 0,Y 558.869,Z 319.37,A -85,B 0,C 180,E1 -2964.589,E2 -2964.589} C_VEL
LIN {X 0,Y 558.868,Z 323.68,A -85,B 0,C 180,E1 -2965.674,E2 -2965.674} C_VEL
LIN {X 0,Y 558.836,Z 325.96,A -85,B 0,C 180,E1 -2966.396,E2 -2966.396} C_VEL
LIN {X 0,Y 558.799,Z 327.809,A -85,B 0,C 180,E1 -2967.117,E2 -2967.117} C_VEL
LIN {X 0,Y 558.745,Z 330.184,A -85,B 0,C 180,E1 -2968.559,E2 -2968.559} C_VEL
LIN {X 0,Y 558.74,Z 331,A -85,B 0,C 180,E1 -2970,E2 -2970} C_VEL
LIN {X 0,Y 558.745,Z 330.184,A -85,B 0,C 180,E1 -2971.442,E2 -2971.442} C_VEL
LIN {X 0,Y 558.799,Z 327.809,A -85,B 0,C 180,E1 -2972.884,E2 -2972.884} C_VEL
LIN {X 0,Y 558.844,Z 324.895,A -85,B 0,C 180,E1 -2973.966,E2 -2973.966} C_VEL
LIN {X 0,Y 558.798,Z 320.948,A -85,B 0,C 180,E1 -2975.051,E2 -2975.051} C_VEL
LIN {X 0,Y 558.919,Z 315.867,A -85,B 0,C 180,E1 -2976.136,E2 -2976.136} C_VEL
LIN {X 0,Y 558.977,Z 309.467,A -85,B 0,C 180,E1 -2977.223,E2 -2977.223} C_VEL
LIN {X 0,Y 559.099,Z 301.478,A -85,B 0,C 180,E1 -2978.312,E2 -2978.312} C_VEL
LIN {X 0,Y 559.194,Z 293.336,A -85,B 0,C 180,E1 -2979.221,E2 -2979.221} C_VEL
LIN {X 0,Y 559.345,Z 283.401,A -85,B 0,C 180,E1 -2980.131,E2 -2980.131} C_VEL
LIN {X 0,Y 559.472,Z 272.448,A -85,B 0,C 180,E1 -2980.935,E2 -2980.935} C_VEL
LIN {X 0,Y 559.635,Z 260.823,A -85,B 0,C 180,E1 -2981.61,E2 -2981.61} C_VEL
LIN {X 0,Y 559.793,Z 248.988,A -85,B 0,C 180,E1 -2982.139,E2 -2982.139} C_VEL
LIN {X 0,Y 559.959,Z 236.191,A -85,B 0,C 180,E1 -2982.549,E2 -2982.549} C_VEL
LIN {X 0,Y 559.818,Z 230.383,A -85,B 0,C 180,E1 -2982.691,E2 -2982.691} C_VEL
LIN {X 0,Y 558.884,Z 224.493,A -85,B 0,C 180,E1 -2982.828,E2 -2982.828} C_VEL
LIN {X 0,Y 558.939,Z 217.05,A -85,B 0,C 180,E1 -2985.31,E2 -2985.31} C_VEL
LIN {X 0,Y 559.004,Z 209.159,A -85,B 0,C 180,E1 -2987.939,E2 -2987.939} C_VEL
LIN {X 0,Y 559.037,Z 201.223,A -85,B 0,C 180,E1 -2990.609,E2 -2990.609} C_VEL
LIN {X 0,Y 559.164,Z 192.223,A -85,B 0,C 180,E1 -2993.715,E2 -2993.715} C_VEL
LIN {X 0,Y 559.211,Z 184.419,A -85,B 0,C 180,E1 -2996.465,E2 -2996.465} C_VEL
LIN {X 0,Y 559.318,Z 177.604,A -85,B 0,C 180,E1 -2998.93,E2 -2998.93} C_VEL
LIN {X 0,Y 559.41,Z 169.804,A -85,B 0,C 180,E1 -3001.845,E2 -3001.845} C_VEL
LIN {X 0,Y 559.51,Z 163.237,A -85,B 0,C 180,E1 -3004.417,E2 -3004.417} C_VEL
LIN {X 0,Y 559.473,Z 159.982,A -85,B 0,C 180,E1 -3005.739,E2 -3005.739} C_VEL
LIN {X 0,Y 559.148,Z 157.84,A -85,B 0,C 180,E1 -3006.745,E2 -3006.745} C_VEL
LIN {X 0,Y 559.168,Z 157.836,A -85,B 0,C 180,E1 -3009.864,E2 -3009.864} C_VEL
LIN {X 0,Y 559.159,Z 157.831,A -85,B 0,C 180,E1 -3012.74,E2 -3012.74} C_VEL
LIN {X 0,Y 559.139,Z 157.835,A -85,B 0,C 180,E1 -3015.759,E2 -3015.759} C_VEL
LIN {X 0,Y 559.149,Z 157.835,A -85,B 0,C 180,E1 -3018.228,E2 -3018.228} C_VEL
LIN {X 0,Y 559.156,Z 157.832,A -85,B 0,C 180,E1 -3021.19,E2 -3021.19} C_VEL
LIN {X 0,Y 559.152,Z 157.837,A -85,B 0,C 180,E1 -3023.79,E2 -3023.79} C_VEL
LIN {X 0,Y 559.157,Z 157.832,A -85,B 0,C 180,E1 -3026.425,E2 -3026.425} C_VEL
LIN {X 0,Y 559.146,Z 157.837,A -85,B 0,C 180,E1 -3028.98,E2 -3028.98} C_VEL
LIN {X 0,Y 559.144,Z 157.835,A -85,B 0,C 180,E1 -3031.617,E2 -3031.617} C_VEL
LIN {X 0,Y 559.148,Z 157.833,A -85,B 0,C 180,E1 -3034.701,E2 -3034.701} C_VEL
LIN {X 0,Y 559.156,Z 157.838,A -85,B 0,C 180,E1 -3037.068,E2 -3037.068} C_VEL
LIN {X 0,Y 559.165,Z 157.831,A -85,B 0,C 180,E1 -3039.395,E2 -3039.395} C_VEL
LIN {X 0,Y 559.184,Z 157.832,A -85,B 0,C 180,E1 -3042.444,E2 -3042.444} C_VEL
LIN {X 0,Y 559.164,Z 157.837,A -85,B 0,C 180,E1 -3045.441,E2 -3045.441} C_VEL
LIN {X 0,Y 559.206,Z 157.828,A -85,B 0,C 180,E1 -3048.587,E2 -3048.587} C_VEL
LIN {X 0,Y 559.183,Z 157.828,A -85,B 0,C 180,E1 -3051.326,E2 -3051.326} C_VEL
LIN {X 0,Y 559.185,Z 157.83,A -85,B 0,C 180,E1 -3053.505,E2 -3053.505} C_VEL
LIN {X 0,Y 559.129,Z 157.841,A -85,B 0,C 180,E1 -3055.675,E2 -3055.675} C_VEL
LIN {X 0,Y 559.214,Z 157.826,A -85,B 0,C 180,E1 -3057.839,E2 -3057.839} C_VEL
LIN {X 0,Y 559.254,Z 157.825,A -85,B 0,C 180,E1 -3060.72,E2 -3060.72} C_VEL
LIN {X 0,Y 559.225,Z 157.824,A -85,B 0,C 180,E1 -3062.882,E2 -3062.882} C_VEL
LIN {X 0,Y 559.222,Z 157.83,A -85,B 0,C 180,E1 -3065.77,E2 -3065.77} C_VEL
LIN {X 0,Y 559.178,Z 157.831,A -85,B 0,C 180,E1 -3068.675,E2 -3068.675} C_VEL
LIN {X 0,Y 559.175,Z 157.83,A -85,B 0,C 180,E1 -3071.601,E2 -3071.601} C_VEL
LIN {X 0,Y 559.169,Z 157.831,A -85,B 0,C 180,E1 -3074.597,E2 -3074.597} C_VEL
LIN {X 0,Y 559.186,Z 157.834,A -85,B 0,C 180,E1 -3077.556,E2 -3077.556} C_VEL
LIN {X 0,Y 559.166,Z 157.834,A -85,B 0,C 180,E1 -3080.605,E2 -3080.605} C_VEL
LIN {X 0,Y 559.122,Z 157.838,A -85,B 0,C 180,E1 -3083.718,E2 -3083.718} C_VEL
LIN {X 0,Y 559.173,Z 157.834,A -85,B 0,C 180,E1 -3086.098,E2 -3086.098} C_VEL
LIN {X 0,Y 559.143,Z 157.833,A -85,B 0,C 180,E1 -3088.531,E2 -3088.531} C_VEL
LIN {X 0,Y 559.134,Z 157.836,A -85,B 0,C 180,E1 -3090.648,E2 -3090.648} C_VEL
LIN {X 0,Y 558.473,Z 157.923,A -85,B 0,C 180,E1 -3091.249,E2 -3091.249} C_VEL
LIN {X 0,Y 555.609,Z 158.277,A -85,B 0,C 180,E1 -3092.225,E2 -3092.225} C_VEL
LIN {X 0,Y 553.195,Z 158.577,A -85,B 0,C 180,E1 -3093.011,E2 -3093.011} C_VEL
LIN {X 0,Y 552.175,Z 158.702,A -85,B 0,C 180,E1 -3093.618,E2 -3093.618} C_VEL
LIN {X 0,Y 552.101,Z 158.712,A -85,B 0,C 180,E1 -3093.823,E2 -3093.823} C_VEL
LIN {X 0,Y 552.089,Z 158.713,A -85,B 0,C 180,E1 -3096.749,E2 -3096.749} C_VEL
LIN {X 0,Y 552.116,Z 158.713,A -85,B 0,C 180,E1 -3099.529,E2 -3099.529} C_VEL
LIN {X 0,Y 552.116,Z 158.711,A -85,B 0,C 180,E1 -3102.427,E2 -3102.427} C_VEL
LIN {X 0,Y 552.085,Z 158.714,A -85,B 0,C 180,E1 -3105.565,E2 -3105.565} C_VEL
LIN {X 0,Y 552.118,Z 158.709,A -85,B 0,C 180,E1 -3108.557,E2 -3108.557} C_VEL
LIN {X 0,Y 552.099,Z 158.715,A -85,B 0,C 180,E1 -3111.412,E2 -3111.412} C_VEL
LIN {X 0,Y 552.038,Z 158.721,A -85,B 0,C 180,E1 -3112.334,E2 -3112.334} C_VEL
LIN {X 0,Y 552.027,Z 159.733,A -85,B 0,C 180,E1 -3113.329,E2 -3113.329} C_VEL
LIN {X 0,Y 552.013,Z 163.865,A -85,B 0,C 180,E1 -3115.933,E2 -3115.933} C_VEL
LIN {X 0,Y 551.997,Z 168.081,A -85,B 0,C 180,E1 -3118.545,E2 -3118.545} C_VEL
LIN {X 0,Y 551.958,Z 172.915,A -85,B 0,C 180,E1 -3121.471,E2 -3121.471} C_VEL
LIN {X 0,Y 551.901,Z 178.39,A -85,B 0,C 180,E1 -3124.707,E2 -3124.707} C_VEL
LIN {X 0,Y 551.796,Z 183.261,A -85,B 0,C 180,E1 -3127.538,E2 -3127.538} C_VEL
LIN {X 0,Y 551.795,Z 188.728,A -85,B 0,C 180,E1 -3130.662,E2 -3130.662} C_VEL
LIN {X 0,Y 551.705,Z 194.158,A -85,B 0,C 180,E1 -3133.726,E2 -3133.726} C_VEL
LIN {X 0,Y 551.662,Z 196.574,A -85,B 0,C 180,E1 -3135.07,E2 -3135.07} C_VEL
LIN {X 0,Y 553.069,Z 206.184,A -85,B 0,C 180,E1 -3135.336,E2 -3135.336} C_VEL
LIN {X 0,Y 552.892,Z 218.476,A -85,B 0,C 180,E1 -3135.732,E2 -3135.732} C_VEL
LIN {X 0,Y 552.66,Z 231.069,A -85,B 0,C 180,E1 -3136.3,E2 -3136.3} C_VEL
LIN {X 0,Y 552.438,Z 242.153,A -85,B 0,C 180,E1 -3136.95,E2 -3136.95} C_VEL
LIN {X 0,Y 552.334,Z 253.445,A -85,B 0,C 180,E1 -3137.788,E2 -3137.788} C_VEL
LIN {X 0,Y 552.145,Z 263.307,A -85,B 0,C 180,E1 -3138.702,E2 -3138.702} C_VEL
LIN {X 0,Y 552.037,Z 272.34,A -85,B 0,C 180,E1 -3139.733,E2 -3139.733} C_VEL
LIN {X 0,Y 551.918,Z 280.186,A -85,B 0,C 180,E1 -3140.841,E2 -3140.841} C_VEL
LIN {X 0,Y 551.826,Z 286.444,A -85,B 0,C 180,E1 -3141.947,E2 -3141.947} C_VEL
LIN {X 0,Y 551.816,Z 291.416,A -85,B 0,C 180,E1 -3143.051,E2 -3143.051} C_VEL
LIN {X 0,Y 551.758,Z 295.255,A -85,B 0,C 180,E1 -3144.151,E2 -3144.151} C_VEL
LIN {X 0,Y 551.695,Z 297.231,A -85,B 0,C 180,E1 -3144.884,E2 -3144.884} C_VEL
LIN {X 0,Y 551.703,Z 298.792,A -85,B 0,C 180,E1 -3145.616,E2 -3145.616} C_VEL
LIN {X 0,Y 551.733,Z 299.924,A -85,B 0,C 180,E1 -3146.348,E2 -3146.348} C_VEL
LIN {X 0,Y 551.719,Z 300.631,A -85,B 0,C 180,E1 -3147.079,E2 -3147.079} C_VEL
LIN {X 0,Y 551.644,Z 300.898,A -85,B 0,C 180,E1 -3148.54,E2 -3148.54} C_VEL
LIN {X 0,Y 551.641,Z 300.438,A -85,B 0,C 180,E1 -3149.27,E2 -3149.27} C_VEL
LIN {X 0,Y 551.645,Z 298.283,A -85,B 0,C 180,E1 -3150.729,E2 -3150.729} C_VEL
LIN {X 0,Y 551.744,Z 295.587,A -85,B 0,C 180,E1 -3151.824,E2 -3151.824} C_VEL
LIN {X 0,Y 551.752,Z 291.885,A -85,B 0,C 180,E1 -3152.92,E2 -3152.92} C_VEL
LIN {X 0,Y 551.822,Z 287.073,A -85,B 0,C 180,E1 -3154.016,E2 -3154.016} C_VEL
LIN {X 0,Y 551.899,Z 281.009,A -85,B 0,C 180,E1 -3155.113,E2 -3155.113} C_VEL
LIN {X 0,Y 552.03,Z 273.479,A -85,B 0,C 180,E1 -3156.211,E2 -3156.211} C_VEL
LIN {X 0,Y 552.106,Z 265.794,A -85,B 0,C 180,E1 -3157.128,E2 -3157.128} C_VEL
LIN {X 0,Y 552.295,Z 255.357,A -85,B 0,C 180,E1 -3158.137,E2 -3158.137} C_VEL
LIN {X 0,Y 552.463,Z 244.744,A -85,B 0,C 180,E1 -3158.964,E2 -3158.964} C_VEL
LIN {X 0,Y 552.598,Z 234.489,A -85,B 0,C 180,E1 -3159.608,E2 -3159.608} C_VEL
LIN {X 0,Y 552.821,Z 222.256,A -85,B 0,C 180,E1 -3160.205,E2 -3160.205} C_VEL
LIN {X 0,Y 552.957,Z 209.394,A -85,B 0,C 180,E1 -3160.665,E2 -3160.665} C_VEL
LIN {X 0,Y 552.899,Z 203.881,A -85,B 0,C 180,E1 -3160.817,E2 -3160.817} C_VEL
LIN {X 0,Y 551.733,Z 196.58,A -85,B 0,C 180,E1 -3161.014,E2 -3161.014} C_VEL
LIN {X 0,Y 551.756,Z 191.23,A -85,B 0,C 180,E1 -3164.004,E2 -3164.004} C_VEL
LIN {X 0,Y 551.811,Z 185.612,A -85,B 0,C 180,E1 -3167.21,E2 -3167.21} C_VEL
LIN {X 0,Y 551.823,Z 180.567,A -85,B 0,C 180,E1 -3170.111,E2 -3170.111} C_VEL
LIN {X 0,Y 551.891,Z 176.565,A -85,B 0,C 180,E1 -3172.457,E2 -3172.457} C_VEL
LIN {X 0,Y 551.937,Z 171.189,A -85,B 0,C 180,E1 -3175.651,E2 -3175.651} C_VEL
LIN {X 0,Y 552.005,Z 166.439,A -85,B 0,C 180,E1 -3178.538,E2 -3178.538} C_VEL
LIN {X 0,Y 552.035,Z 161.699,A -85,B 0,C 180,E1 -3181.462,E2 -3181.462} C_VEL
LIN {X 0,Y 551.98,Z 158.926,A -85,B 0,C 180,E1 -3183.192,E2 -3183.192} C_VEL
LIN {X 0,Y 552.066,Z 158.721,A -85,B 0,C 180,E1 -3184.947,E2 -3184.947} C_VEL
LIN {X 0,Y 552.079,Z 158.714,A -85,B 0,C 180,E1 -3187.882,E2 -3187.882} C_VEL
LIN {X 0,Y 552.105,Z 158.714,A -85,B 0,C 180,E1 -3190.477,E2 -3190.477} C_VEL
LIN {X 0,Y 552.1,Z 158.715,A -85,B 0,C 180,E1 -3193.482,E2 -3193.482} C_VEL
LIN {X 0,Y 552.103,Z 158.71,A -85,B 0,C 180,E1 -3196.575,E2 -3196.575} C_VEL
LIN {X 0,Y 552.121,Z 158.708,A -85,B 0,C 180,E1 -3199.519,E2 -3199.519} C_VEL
LIN {X 0,Y 552.067,Z 158.72,A -85,B 0,C 180,E1 -3202.334,E2 -3202.334} C_VEL
LIN {X 0,Y 552.091,Z 158.712,A -85,B 0,C 180,E1 -3205.051,E2 -3205.051} C_VEL
LIN {X 0,Y 552.102,Z 158.716,A -85,B 0,C 180,E1 -3207.68,E2 -3207.68} C_VEL
LIN {X 0,Y 552.122,Z 158.708,A -85,B 0,C 180,E1 -3210.235,E2 -3210.235} C_VEL
LIN {X 0,Y 552.129,Z 158.712,A -85,B 0,C 180,E1 -3212.993,E2 -3212.993} C_VEL
LIN {X 0,Y 552.104,Z 158.71,A -85,B 0,C 180,E1 -3215.16,E2 -3215.16} C_VEL
LIN {X 0,Y 552.093,Z 158.712,A -85,B 0,C 180,E1 -3217.549,E2 -3217.549} C_VEL
LIN {X 0,Y 552.119,Z 158.708,A -85,B 0,C 180,E1 -3220.673,E2 -3220.673} C_VEL
LIN {X 0,Y 552.099,Z 158.713,A -85,B 0,C 180,E1 -3223.736,E2 -3223.736} C_VEL
LIN {X 0,Y 552.112,Z 158.709,A -85,B 0,C 180,E1 -3226.004,E2 -3226.004} C_VEL
LIN {X 0,Y 552.189,Z 158.701,A -85,B 0,C 180,E1 -3228.994,E2 -3228.994} C_VEL
LIN {X 0,Y 552.168,Z 158.707,A -85,B 0,C 180,E1 -3231.951,E2 -3231.951} C_VEL
LIN {X 0,Y 552.21,Z 158.697,A -85,B 0,C 180,E1 -3234.889,E2 -3234.889} C_VEL
LIN {X 0,Y 552.18,Z 158.702,A -85,B 0,C 180,E1 -3237.812,E2 -3237.812} C_VEL
LIN {X 0,Y 552.214,Z 158.702,A -85,B 0,C 180,E1 -3240.729,E2 -3240.729} C_VEL
LIN {X 0,Y 552.185,Z 158.703,A -85,B 0,C 180,E1 -3242.918,E2 -3242.918} C_VEL
LIN {X 0,Y 552.188,Z 158.705,A -85,B 0,C 180,E1 -3245.844,E2 -3245.844} C_VEL
LIN {X 0,Y 552.146,Z 158.704,A -85,B 0,C 180,E1 -3248.786,E2 -3248.786} C_VEL
LIN {X 0,Y 552.13,Z 158.708,A -85,B 0,C 180,E1 -3251.751,E2 -3251.751} C_VEL
LIN {X 0,Y 552.097,Z 158.717,A -85,B 0,C 180,E1 -3254.749,E2 -3254.749} C_VEL
LIN {X 0,Y 552.077,Z 158.716,A -85,B 0,C 180,E1 -3257.79,E2 -3257.79} C_VEL
LIN {X 0,Y 552.1,Z 158.716,A -85,B 0,C 180,E1 -3260.102,E2 -3260.102} C_VEL
LIN {X 0,Y 552.122,Z 158.712,A -85,B 0,C 180,E1 -3263.241,E2 -3263.241} C_VEL
LIN {X 0,Y 552.142,Z 158.706,A -85,B 0,C 180,E1 -3265.644,E2 -3265.644} C_VEL
LIN {X 0,Y 552.113,Z 158.714,A -85,B 0,C 180,E1 -3268.568,E2 -3268.568} C_VEL
LIN {X 0,Y 552.104,Z 158.71,A -85,B 0,C 180,E1 -3271.482,E2 -3271.482} C_VEL
LIN {X 0,Y 552.104,Z 158.714,A -85,B 0,C 180,E1 -3274.173,E2 -3274.173} C_VEL
LIN {X 0,Y 552.083,Z 158.713,A -85,B 0,C 180,E1 -3276.749,E2 -3276.749} C_VEL
LIN {X 0,Y 552.112,Z 158.712,A -85,B 0,C 180,E1 -3279.529,E2 -3279.529} C_VEL
LIN {X 0,Y 552.149,Z 158.705,A -85,B 0,C 180,E1 -3281.443,E2 -3281.443} C_VEL
LIN {X 0,Y 552.075,Z 158.718,A -85,B 0,C 180,E1 -3284.535,E2 -3284.535} C_VEL
LIN {X 0,Y 552.113,Z 158.714,A -85,B 0,C 180,E1 -3287.587,E2 -3287.587} C_VEL
LIN {X 0,Y 552.11,Z 158.711,A -85,B 0,C 180,E1 -3290.475,E2 -3290.475} C_VEL
LIN {X 0,Y 552.136,Z 158.811,A -85,B 0,C 180,E1 -3293.313,E2 -3293.313} C_VEL
LIN {X 0,Y 552.519,Z 163.069,A -85,B 0,C 180,E1 -3295.086,E2 -3295.086} C_VEL
LIN {X 0,Y 552.385,Z 169.701,A -85,B 0,C 180,E1 -3297.702,E2 -3297.702} C_VEL
LIN {X 0,Y 552.327,Z 177.533,A -85,B 0,C 180,E1 -3300.67,E2 -3300.67} C_VEL
LIN {X 0,Y 552.173,Z 185.375,A -85,B 0,C 180,E1 -3303.549,E2 -3303.549} C_VEL
LIN {X 0,Y 552.133,Z 192.111,A -85,B 0,C 180,E1 -3305.966,E2 -3305.966} C_VEL
LIN {X 0,Y 551.996,Z 201.11,A -85,B 0,C 180,E1 -3309.117,E2 -3309.117} C_VEL
LIN {X 0,Y 551.932,Z 208.974,A -85,B 0,C 180,E1 -3311.824,E2 -3311.824} C_VEL
LIN {X 0,Y 551.863,Z 216.932,A -85,B 0,C 180,E1 -3314.49,E2 -3314.49} C_VEL
LIN {X 0,Y 551.798,Z 224.496,A -85,B 0,C 180,E1 -3317.006,E2 -3317.006} C_VEL
LIN {X 0,Y 553.072,Z 233.492,A -85,B 0,C 180,E1 -3317.223,E2 -3317.223} C_VEL
LIN {X 0,Y 552.899,Z 246.514,A -85,B 0,C 180,E1 -3317.615,E2 -3317.615} C_VEL
LIN {X 0,Y 552.738,Z 257.519,A -85,B 0,C 180,E1 -3318.077,E2 -3318.077} C_VEL
LIN {X 0,Y 552.551,Z 269.396,A -85,B 0,C 180,E1 -3318.728,E2 -3318.728} C_VEL
LIN {X 0,Y 552.41,Z 281.108,A -85,B 0,C 180,E1 -3319.556,E2 -3319.556} C_VEL
LIN {X 0,Y 552.199,Z 291.552,A -85,B 0,C 180,E1 -3320.478,E2 -3320.478} C_VEL
LIN {X 0,Y 552.081,Z 300.001,A -85,B 0,C 180,E1 -3321.399,E2 -3321.399} C_VEL
LIN {X 0,Y 551.925,Z 308.242,A -85,B 0,C 180,E1 -3322.501,E2 -3322.501} C_VEL
LIN {X 0,Y 551.82,Z 315.211,A -85,B 0,C 180,E1 -3323.663,E2 -3323.663} C_VEL
LIN {X 0,Y 551.723,Z 320.953,A -85,B 0,C 180,E1 -3324.885,E2 -3324.885} C_VEL
LIN {X 0,Y 551.763,Z 324.897,A -85,B 0,C 180,E1 -3325.984,E2 -3325.984} C_VEL
LIN {X 0,Y 551.723,Z 327.809,A -85,B 0,C 180,E1 -3327.08,E2 -3327.08} C_VEL
LIN {X 0,Y 551.645,Z 330.184,A -85,B 0,C 180,E1 -3328.541,E2 -3328.541} C_VEL
LIN {X 0,Y 551.64,Z 331,A -85,B 0,C 180,E1 -3330,E2 -3330} C_VEL
LIN {X 0,Y 551.645,Z 330.184,A -85,B 0,C 180,E1 -3331.46,E2 -3331.46} C_VEL
LIN {X 0,Y 551.723,Z 327.809,A -85,B 0,C 180,E1 -3332.921,E2 -3332.921} C_VEL
LIN {X 0,Y 551.764,Z 324.895,A -85,B 0,C 180,E1 -3334.017,E2 -3334.017} C_VEL
LIN {X 0,Y 551.723,Z 320.948,A -85,B 0,C 180,E1 -3335.116,E2 -3335.116} C_VEL
LIN {X 0,Y 551.814,Z 315.127,A -85,B 0,C 180,E1 -3336.353,E2 -3336.353} C_VEL
LIN {X 0,Y 551.926,Z 308.236,A -85,B 0,C 180,E1 -3337.5,E2 -3337.5} C_VEL
LIN {X 0,Y 552.082,Z 299.993,A -85,B 0,C 180,E1 -3338.602,E2 -3338.602} C_VEL
LIN {X 0,Y 552.2,Z 291.542,A -85,B 0,C 180,E1 -3339.523,E2 -3339.523} C_VEL
LIN {X 0,Y 552.41,Z 281.095,A -85,B 0,C 180,E1 -3340.445,E2 -3340.445} C_VEL
LIN {X 0,Y 552.55,Z 269.35,A -85,B 0,C 180,E1 -3341.276,E2 -3341.276} C_VEL
LIN {X 0,Y 552.742,Z 257.494,A -85,B 0,C 180,E1 -3341.924,E2 -3341.924} C_VEL
LIN {X 0,Y 552.956,Z 245.175,A -85,B 0,C 180,E1 -3342.431,E2 -3342.431} C_VEL
LIN {X 0,Y 553.032,Z 232.052,A -85,B 0,C 180,E1 -3342.814,E2 -3342.814} C_VEL
LIN {X 0,Y 551.795,Z 224.493,A -85,B 0,C 180,E1 -3342.995,E2 -3342.995} C_VEL
LIN {X 0,Y 551.891,Z 215.817,A -85,B 0,C 180,E1 -3345.889,E2 -3345.889} C_VEL
LIN {X 0,Y 551.962,Z 206.749,A -85,B 0,C 180,E1 -3348.946,E2 -3348.946} C_VEL
LIN {X 0,Y 552.042,Z 198.853,A -85,B 0,C 180,E1 -3351.665,E2 -3351.665} C_VEL
LIN {X 0,Y 552.117,Z 190.968,A -85,B 0,C 180,E1 -3354.436,E2 -3354.436} C_VEL
LIN {X 0,Y 552.198,Z 183.11,A -85,B 0,C 180,E1 -3357.268,E2 -3357.268} C_VEL
LIN {X 0,Y 552.325,Z 175.52,A -85,B 0,C 180,E1 -3360.087,E2 -3360.087} C_VEL
LIN {X 0,Y 552.508,Z 167.562,A -85,B 0,C 180,E1 -3363.157,E2 -3363.157} C_VEL
LIN {X 0,Y 552.476,Z 161.05,A -85,B 0,C 180,E1 -3365.812,E2 -3365.812} C_VEL
LIN {X 0,Y 552.12,Z 158.715,A -85,B 0,C 180,E1 -3366.857,E2 -3366.857} C_VEL
LIN {X 0,Y 552.117,Z 158.712,A -85,B 0,C 180,E1 -3369.525,E2 -3369.525} C_VEL
LIN {X 0,Y 552.119,Z 158.709,A -85,B 0,C 180,E1 -3372.423,E2 -3372.423} C_VEL
LIN {X 0,Y 552.084,Z 158.716,A -85,B 0,C 180,E1 -3375.561,E2 -3375.561} C_VEL
LIN {X 0,Y 552.105,Z 158.715,A -85,B 0,C 180,E1 -3378.553,E2 -3378.553} C_VEL
LIN {X 0,Y 552.098,Z 158.712,A -85,B 0,C 180,E1 -3381.409,E2 -3381.409} C_VEL
LIN {X 0,Y 552.094,Z 158.712,A -85,B 0,C 180,E1 -3384.157,E2 -3384.157} C_VEL
LIN {X 0,Y 552.108,Z 158.713,A -85,B 0,C 180,E1 -3386.814,E2 -3386.814} C_VEL
LIN {X 0,Y 552.092,Z 158.712,A -85,B 0,C 180,E1 -3389.39,E2 -3389.39} C_VEL
LIN {X 0,Y 552.099,Z 158.716,A -85,B 0,C 180,E1 -3391.901,E2 -3391.901} C_VEL
LIN {X 0,Y 552.128,Z 158.708,A -85,B 0,C 180,E1 -3394.648,E2 -3394.648} C_VEL
LIN {X 0,Y 552.102,Z 158.711,A -85,B 0,C 180,E1 -3397.549,E2 -3397.549} C_VEL
LIN {X 0,Y 552.131,Z 158.712,A -85,B 0,C 180,E1 -3400.674,E2 -3400.674} C_VEL
LIN {X 0,Y 552.165,Z 158.703,A -85,B 0,C 180,E1 -3402.978,E2 -3402.978} C_VEL
LIN {X 0,Y 552.105,Z 158.712,A -85,B 0,C 180,E1 -3406.004,E2 -3406.004} C_VEL
LIN {X 0,Y 552.184,Z 158.705,A -85,B 0,C 180,E1 -3408.994,E2 -3408.994} C_VEL
LIN {X 0,Y 552.148,Z 158.707,A -85,B 0,C 180,E1 -3411.952,E2 -3411.952} C_VEL
LIN {X 0,Y 552.194,Z 158.704,A -85,B 0,C 180,E1 -3414.156,E2 -3414.156} C_VEL
LIN {X 0,Y 552.183,Z 158.705,A -85,B 0,C 180,E1 -3417.082,E2 -3417.082} C_VEL
LIN {X 0,Y 552.192,Z 158.7,A -85,B 0,C 180,E1 -3420,E2 -3420} C_VEL
LIN {X 0,Y 552.191,Z 158.7,A -85,B 0,C 180,E1 -3422.918,E2 -3422.918} C_VEL
LIN {X 0,Y 552.191,Z 158.705,A -85,B 0,C 180,E1 -3425.844,E2 -3425.844} C_VEL
LIN {X 0,Y 552.145,Z 158.709,A -85,B 0,C 180,E1 -3428.786,E2 -3428.786} C_VEL
LIN {X 0,Y 552.132,Z 158.707,A -85,B 0,C 180,E1 -3431.751,E2 -3431.751} C_VEL
LIN {X 0,Y 552.109,Z 158.71,A -85,B 0,C 180,E1 -3434.749,E2 -3434.749} C_VEL
LIN {X 0,Y 552.118,Z 158.712,A -85,B 0,C 180,E1 -3437.789,E2 -3437.789} C_VEL
LIN {X 0,Y 552.111,Z 158.71,A -85,B 0,C 180,E1 -3440.102,E2 -3440.102} C_VEL
LIN {X 0,Y 552.076,Z 158.719,A -85,B 0,C 180,E1 -3442.452,E2 -3442.452} C_VEL
LIN {X 0,Y 552.131,Z 158.708,A -85,B 0,C 180,E1 -3445.352,E2 -3445.352} C_VEL
LIN {X 0,Y 552.104,Z 158.711,A -85,B 0,C 180,E1 -3448.099,E2 -3448.099} C_VEL
LIN {X 0,Y 552.093,Z 158.713,A -85,B 0,C 180,E1 -3450.643,E2 -3450.643} C_VEL
LIN {X 0,Y 552.109,Z 158.711,A -85,B 0,C 180,E1 -3453.187,E2 -3453.187} C_VEL
LIN {X 0,Y 552.101,Z 158.712,A -85,B 0,C 180,E1 -3453.823,E2 -3453.823} C_VEL
LIN {X 0,Y 551.466,Z 158.796,A -85,B 0,C 180,E1 -3454.432,E2 -3454.432} C_VEL
LIN {X 0,Y 548.639,Z 159.145,A -85,B 0,C 180,E1 -3455.42,E2 -3455.42} C_VEL
LIN {X 0,Y 546.213,Z 159.449,A -85,B 0,C 180,E1 -3456.215,E2 -3456.215} C_VEL
LIN {X 0,Y 545.142,Z 159.579,A -85,B 0,C 180,E1 -3456.829,E2 -3456.829} C_VEL
LIN {X 0,Y 545.041,Z 159.591,A -85,B 0,C 180,E1 -3457.037,E2 -3457.037} C_VEL
LIN {X 0,Y 545.058,Z 159.588,A -85,B 0,C 180,E1 -3460.144,E2 -3460.144} C_VEL
LIN {X 0,Y 545.049,Z 159.595,A -85,B 0,C 180,E1 -3462.699,E2 -3462.699} C_VEL
LIN {X 0,Y 545.049,Z 159.589,A -85,B 0,C 180,E1 -3465.169,E2 -3465.169} C_VEL
LIN {X 0,Y 545.069,Z 159.592,A -85,B 0,C 180,E1 -3467.899,E2 -3467.899} C_VEL
LIN {X 0,Y 545.066,Z 159.59,A -85,B 0,C 180,E1 -3470.82,E2 -3470.82} C_VEL
LIN {X 0,Y 544.952,Z 159.618,A -85,B 0,C 180,E1 -3472.692,E2 -3472.692} C_VEL
LIN {X 0,Y 544.968,Z 164.204,A -85,B 0,C 180,E1 -3475.625,E2 -3475.625} C_VEL
LIN {X 0,Y 544.93,Z 168.531,A -85,B 0,C 180,E1 -3478.344,E2 -3478.344} C_VEL
LIN {X 0,Y 544.911,Z 173.674,A -85,B 0,C 180,E1 -3481.498,E2 -3481.498} C_VEL
LIN {X 0,Y 544.854,Z 179.231,A -85,B 0,C 180,E1 -3484.809,E2 -3484.809} C_VEL
LIN {X 0,Y 544.723,Z 183.351,A -85,B 0,C 180,E1 -3487.23,E2 -3487.23} C_VEL
LIN {X 0,Y 544.736,Z 188.882,A -85,B 0,C 180,E1 -3490.401,E2 -3490.401} C_VEL
LIN {X 0,Y 544.631,Z 194.3,A -85,B 0,C 180,E1 -3493.508,E2 -3493.508} C_VEL
LIN {X 0,Y 544.606,Z 196.827,A -85,B 0,C 180,E1 -3494.915,E2 -3494.915} C_VEL
LIN {X 0,Y 546.143,Z 206.753,A -85,B 0,C 180,E1 -3495.182,E2 -3495.182} C_VEL
LIN {X 0,Y 545.955,Z 218.882,A -85,B 0,C 180,E1 -3495.582,E2 -3495.582} C_VEL
LIN {X 0,Y 545.739,Z 230.74,A -85,B 0,C 180,E1 -3496.123,E2 -3496.123} C_VEL
LIN {X 0,Y 545.467,Z 241.89,A -85,B 0,C 180,E1 -3496.78,E2 -3496.78} C_VEL
LIN {X 0,Y 545.353,Z 253.239,A -85,B 0,C 180,E1 -3497.629,E2 -3497.629} C_VEL
LIN {X 0,Y 545.154,Z 262.209,A -85,B 0,C 180,E1 -3498.46,E2 -3498.46} C_VEL
LIN {X 0,Y 545.027,Z 270.668,A -85,B 0,C 180,E1 -3499.412,E2 -3499.412} C_VEL
LIN {X 0,Y 544.83,Z 278.808,A -85,B 0,C 180,E1 -3500.534,E2 -3500.534} C_VEL
LIN {X 0,Y 544.754,Z 284.359,A -85,B 0,C 180,E1 -3501.468,E2 -3501.468} C_VEL
LIN {X 0,Y 544.718,Z 289.777,A -85,B 0,C 180,E1 -3502.587,E2 -3502.587} C_VEL
LIN {X 0,Y 544.669,Z 293.305,A -85,B 0,C 180,E1 -3503.494,E2 -3503.494} C_VEL
LIN {X 0,Y 544.616,Z 297.169,A -85,B 0,C 180,E1 -3504.817,E2 -3504.817} C_VEL
LIN {X 0,Y 544.6,Z 298.742,A -85,B 0,C 180,E1 -3505.559,E2 -3505.559} C_VEL
LIN {X 0,Y 544.647,Z 299.896,A -85,B 0,C 180,E1 -3506.301,E2 -3506.301} C_VEL
LIN {X 0,Y 544.646,Z 300.614,A -85,B 0,C 180,E1 -3507.041,E2 -3507.041} C_VEL
LIN {X 0,Y 544.545,Z 300.904,A -85,B 0,C 180,E1 -3508.521,E2 -3508.521} C_VEL
LIN {X 0,Y 544.542,Z 300.464,A -85,B 0,C 180,E1 -3509.26,E2 -3509.26} C_VEL
LIN {X 0,Y 544.546,Z 298.332,A -85,B 0,C 180,E1 -3510.739,E2 -3510.739} C_VEL
LIN {X 0,Y 544.666,Z 295.66,A -85,B 0,C 180,E1 -3511.848,E2 -3511.848} C_VEL
LIN {X 0,Y 544.682,Z 291.983,A -85,B 0,C 180,E1 -3512.958,E2 -3512.958} C_VEL
LIN {X 0,Y 544.743,Z 287.197,A -85,B 0,C 180,E1 -3514.068,E2 -3514.068} C_VEL
LIN {X 0,Y 544.826,Z 281.163,A -85,B 0,C 180,E1 -3515.18,E2 -3515.18} C_VEL
LIN {X 0,Y 544.989,Z 273.764,A -85,B 0,C 180,E1 -3516.28,E2 -3516.28} C_VEL
LIN {X 0,Y 545.063,Z 266.228,A -85,B 0,C 180,E1 -3517.202,E2 -3517.202} C_VEL
LIN {X 0,Y 545.276,Z 256.795,A -85,B 0,C 180,E1 -3518.15,E2 -3518.15} C_VEL
LIN {X 0,Y 545.477,Z 246.497,A -85,B 0,C 180,E1 -3518.986,E2 -3518.986} C_VEL
LIN {X 0,Y 545.643,Z 235.071,A -85,B 0,C 180,E1 -3519.732,E2 -3519.732} C_VEL
LIN {X 0,Y 545.88,Z 223.049,A -85,B 0,C 180,E1 -3520.336,E2 -3520.336} C_VEL
LIN {X 0,Y 546.035,Z 209.667,A -85,B 0,C 180,E1 -3520.825,E2 -3520.825} C_VEL
LIN {X 0,Y 545.946,Z 204.63,A -85,B 0,C 180,E1 -3520.968,E2 -3520.968} C_VEL
LIN {X 0,Y 544.651,Z 196.699,A -85,B 0,C 180,E1 -3521.201,E2 -3521.201} C_VEL
LIN {X 0,Y 544.722,Z 190.678,A -85,B 0,C 180,E1 -3524.612,E2 -3524.612} C_VEL
LIN {X 0,Y 544.742,Z 186.028,A -85,B 0,C 180,E1 -3527.308,E2 -3527.308} C_VEL
LIN {X 0,Y 544.771,Z 180.746,A -85,B 0,C 180,E1 -3530.383,E2 -3530.383} C_VEL
LIN {X 0,Y 544.827,Z 176.717,A -85,B 0,C 180,E1 -3532.765,E2 -3532.765} C_VEL
LIN {X 0,Y 544.865,Z 172.241,A -85,B 0,C 180,E1 -3535.457,E2 -3535.457} C_VEL
LIN {X 0,Y 544.954,Z 167.275,A -85,B 0,C 180,E1 -3538.498,E2 -3538.498} C_VEL
LIN {X 0,Y 545,Z 163.181,A -85,B 0,C 180,E1 -3541.049,E2 -3541.049} C_VEL
LIN {X 0,Y 544.946,Z 160.023,A -85,B 0,C 180,E1 -3543.04,E2 -3543.04} C_VEL
LIN {X 0,Y 544.983,Z 159.601,A -85,B 0,C 180,E1 -3543.674,E2 -3543.674} C_VEL
LIN {X 0,Y 545.021,Z 159.595,A -85,B 0,C 180,E1 -3546.378,E2 -3546.378} C_VEL
LIN {X 0,Y 545.086,Z 159.585,A -85,B 0,C 180,E1 -3549.321,E2 -3549.321} C_VEL
LIN {X 0,Y 545.068,Z 159.591,A -85,B 0,C 180,E1 -3552.1,E2 -3552.1} C_VEL
LIN {X 0,Y 545.044,Z 159.593,A -85,B 0,C 180,E1 -3555.164,E2 -3555.164} C_VEL
LIN {X 0,Y 545.071,Z 159.585,A -85,B 0,C 180,E1 -3557.896,E2 -3557.896} C_VEL
LIN {X 0,Y 545.061,Z 159.593,A -85,B 0,C 180,E1 -3560.816,E2 -3560.816} C_VEL
LIN {X 0,Y 545.022,Z 159.593,A -85,B 0,C 180,E1 -3563.618,E2 -3563.618} C_VEL
LIN {X 0,Y 545.047,Z 159.592,A -85,B 0,C 180,E1 -3566.326,E2 -3566.326} C_VEL
LIN {X 0,Y 545.043,Z 159.592,A -85,B 0,C 180,E1 -3568.95,E2 -3568.95} C_VEL
LIN {X 0,Y 545.091,Z 159.586,A -85,B 0,C 180,E1 -3571.507,E2 -3571.507} C_VEL
LIN {X 0,Y 545.101,Z 159.587,A -85,B 0,C 180,E1 -3574.48,E2 -3574.48} C_VEL
LIN {X 0,Y 545.047,Z 159.589,A -85,B 0,C 180,E1 -3577.242,E2 -3577.242} C_VEL
LIN {X 0,Y 545.084,Z 159.586,A -85,B 0,C 180,E1 -3580.413,E2 -3580.413} C_VEL
LIN {X 0,Y 545.056,Z 159.593,A -85,B 0,C 180,E1 -3583.52,E2 -3583.52} C_VEL
LIN {X 0,Y 545.087,Z 159.588,A -85,B 0,C 180,E1 -3586.58,E2 -3586.58} C_VEL
LIN {X 0,Y 545.16,Z 159.579,A -85,B 0,C 180,E1 -3588.85,E2 -3588.85} C_VEL
LIN {X 0,Y 545.127,Z 159.583,A -85,B 0,C 180,E1 -3591.847,E2 -3591.847} C_VEL
LIN {X 0,Y 545.185,Z 159.572,A -85,B 0,C 180,E1 -3594.823,E2 -3594.823} C_VEL
LIN {X 0,Y 545.153,Z 159.578,A -85,B 0,C 180,E1 -3597.783,E2 -3597.783} C_VEL
LIN {X 0,Y 545.183,Z 159.577,A -85,B 0,C 180,E1 -3600.738,E2 -3600.738} C_VEL
LIN {X 0,Y 545.15,Z 159.579,A -85,B 0,C 180,E1 -3602.956,E2 -3602.956} C_VEL
LIN {X 0,Y 545.159,Z 159.581,A -85,B 0,C 180,E1 -3605.919,E2 -3605.919} C_VEL
LIN {X 0,Y 545.127,Z 159.581,A -85,B 0,C 180,E1 -3608.153,E2 -3608.153} C_VEL
LIN {X 0,Y 545.116,Z 159.583,A -85,B 0,C 180,E1 -3611.547,E2 -3611.547} C_VEL
LIN {X 0,Y 545.063,Z 159.593,A -85,B 0,C 180,E1 -3614.768,E2 -3614.768} C_VEL
LIN {X 0,Y 545.056,Z 159.588,A -85,B 0,C 180,E1 -3617.43,E2 -3617.43} C_VEL
LIN {X 0,Y 545.065,Z 159.59,A -85,B 0,C 180,E1 -3620.373,E2 -3620.373} C_VEL
LIN {X 0,Y 545.116,Z 159.585,A -85,B 0,C 180,E1 -3623.558,E2 -3623.558} C_VEL
LIN {X 0,Y 545.081,Z 159.584,A -85,B 0,C 180,E1 -3626,E2 -3626} C_VEL
LIN {X 0,Y 545.076,Z 159.592,A -85,B 0,C 180,E1 -3628.754,E2 -3628.754} C_VEL
LIN {X 0,Y 545.047,Z 159.591,A -85,B 0,C 180,E1 -3631.685,E2 -3631.685} C_VEL
LIN {X 0,Y 545.047,Z 159.59,A -85,B 0,C 180,E1 -3634.566,E2 -3634.566} C_VEL
LIN {X 0,Y 545.013,Z 159.599,A -85,B 0,C 180,E1 -3637.306,E2 -3637.306} C_VEL
LIN {X 0,Y 545.071,Z 159.586,A -85,B 0,C 180,E1 -3640.142,E2 -3640.142} C_VEL
LIN {X 0,Y 545.046,Z 159.595,A -85,B 0,C 180,E1 -3642.7,E2 -3642.7} C_VEL
LIN {X 0,Y 545.042,Z 159.589,A -85,B 0,C 180,E1 -3645.169,E2 -3645.169} C_VEL
LIN {X 0,Y 545.065,Z 159.594,A -85,B 0,C 180,E1 -3647.9,E2 -3647.9} C_VEL
LIN {X 0,Y 545.06,Z 159.591,A -85,B 0,C 180,E1 -3650.821,E2 -3650.821} C_VEL
LIN {X 0,Y 545.072,Z 159.651,A -85,B 0,C 180,E1 -3653.141,E2 -3653.141} C_VEL
LIN {X 0,Y 545.533,Z 162.999,A -85,B 0,C 180,E1 -3654.572,E2 -3654.572} C_VEL
LIN {X 0,Y 545.409,Z 169.618,A -85,B 0,C 180,E1 -3657.238,E2 -3657.238} C_VEL
LIN {X 0,Y 545.314,Z 177.43,A -85,B 0,C 180,E1 -3660.255,E2 -3660.255} C_VEL
LIN {X 0,Y 545.138,Z 185.277,A -85,B 0,C 180,E1 -3663.18,E2 -3663.18} C_VEL
LIN {X 0,Y 545.066,Z 192.011,A -85,B 0,C 180,E1 -3665.634,E2 -3665.634} C_VEL
LIN {X 0,Y 544.96,Z 200.99,A -85,B 0,C 180,E1 -3668.835,E2 -3668.835} C_VEL
LIN {X 0,Y 544.866,Z 208.828,A -85,B 0,C 180,E1 -3671.58,E2 -3671.58} C_VEL
LIN {X 0,Y 544.804,Z 216.766,A -85,B 0,C 180,E1 -3674.284,E2 -3674.284} C_VEL
LIN {X 0,Y 544.734,Z 224.344,A -85,B 0,C 180,E1 -3676.834,E2 -3676.834} C_VEL
LIN {X 0,Y 546.144,Z 234.269,A -85,B 0,C 180,E1 -3677.082,E2 -3677.082} C_VEL
LIN {X 0,Y 545.943,Z 247.695,A -85,B 0,C 180,E1 -3677.502,E2 -3677.502} C_VEL
LIN {X 0,Y 545.757,Z 259.338,A -85,B 0,C 180,E1 -3678.017,E2 -3678.017} C_VEL
LIN {X 0,Y 545.551,Z 269.698,A -85,B 0,C 180,E1 -3678.606,E2 -3678.606} C_VEL
LIN {X 0,Y 545.403,Z 281.078,A -85,B 0,C 180,E1 -3679.42,E2 -3679.42} C_VEL
LIN {X 0,Y 545.162,Z 291.552,A -85,B 0,C 180,E1 -3680.353,E2 -3680.353} C_VEL
LIN {X 0,Y 545.028,Z 300.001,A -85,B 0,C 180,E1 -3681.287,E2 -3681.287} C_VEL
LIN {X 0,Y 544.858,Z 308.242,A -85,B 0,C 180,E1 -3682.404,E2 -3682.404} C_VEL
LIN {X 0,Y 544.733,Z 315.619,A -85,B 0,C 180,E1 -3683.656,E2 -3683.656} C_VEL
LIN {X 0,Y 544.653,Z 320.953,A -85,B 0,C 180,E1 -3684.819,E2 -3684.819} C_VEL
LIN {X 0,Y 544.683,Z 324.896,A -85,B 0,C 180,E1 -3685.931,E2 -3685.931} C_VEL
LIN {X 0,Y 544.65,Z 327.808,A -85,B 0,C 180,E1 -3687.042,E2 -3687.042} C_VEL
LIN {X 0,Y 544.546,Z 330.183,A -85,B 0,C 180,E1 -3688.522,E2 -3688.522} C_VEL
LIN {X 0,Y 544.541,Z 331,A -85,B 0,C 180,E1 -3690,E2 -3690} C_VEL
LIN {X 0,Y 544.546,Z 330.183,A -85,B 0,C 180,E1 -3691.479,E2 -3691.479} C_VEL
LIN {X 0,Y 544.65,Z 327.809,A -85,B 0,C 180,E1 -3692.959,E2 -3692.959} C_VEL
LIN {X 0,Y 544.684,Z 324.895,A -85,B 0,C 180,E1 -3694.07,E2 -3694.07} C_VEL
LIN {X 0,Y 544.653,Z 320.947,A -85,B 0,C 180,E1 -3695.182,E2 -3695.182} C_VEL
LIN {X 0,Y 544.729,Z 315.647,A -85,B 0,C 180,E1 -3696.339,E2 -3696.339} C_VEL
LIN {X 0,Y 544.836,Z 309.466,A -85,B 0,C 180,E1 -3697.411,E2 -3697.411} C_VEL
LIN {X 0,Y 545.006,Z 301.478,A -85,B 0,C 180,E1 -3698.528,E2 -3698.528} C_VEL
LIN {X 0,Y 545.141,Z 293.334,A -85,B 0,C 180,E1 -3699.461,E2 -3699.461} C_VEL
LIN {X 0,Y 545.359,Z 283.378,A -85,B 0,C 180,E1 -3700.394,E2 -3700.394} C_VEL
LIN {X 0,Y 545.495,Z 273.541,A -85,B 0,C 180,E1 -3701.143,E2 -3701.143} C_VEL
LIN {X 0,Y 545.689,Z 262.543,A -85,B 0,C 180,E1 -3701.814,E2 -3701.814} C_VEL
LIN {X 0,Y 545.879,Z 249.995,A -85,B 0,C 180,E1 -3702.406,E2 -3702.406} C_VEL
LIN {X 0,Y 546.103,Z 236.966,A -85,B 0,C 180,E1 -3702.85,E2 -3702.85} C_VEL
LIN {X 0,Y 545.852,Z 231.226,A -85,B 0,C 180,E1 -3703,E2 -3703} C_VEL
LIN {X 0,Y 544.73,Z 224.366,A -85,B 0,C 180,E1 -3703.167,E2 -3703.167} C_VEL
LIN {X 0,Y 544.806,Z 216.81,A -85,B 0,C 180,E1 -3705.717,E2 -3705.717} C_VEL
LIN {X 0,Y 544.869,Z 208.878,A -85,B 0,C 180,E1 -3708.421,E2 -3708.421} C_VEL
LIN {X 0,Y 544.956,Z 200.978,A -85,B 0,C 180,E1 -3711.167,E2 -3711.167} C_VEL
LIN {X 0,Y 545.057,Z 193.756,A -85,B 0,C 180,E1 -3713.726,E2 -3713.726} C_VEL
LIN {X 0,Y 545.138,Z 186.384,A -85,B 0,C 180,E1 -3716.408,E2 -3716.408} C_VEL
LIN {X 0,Y 545.276,Z 178.566,A -85,B 0,C 180,E1 -3719.324,E2 -3719.324} C_VEL
LIN {X 0,Y 545.397,Z 171.925,A -85,B 0,C 180,E1 -3721.89,E2 -3721.89} C_VEL
LIN {X 0,Y 545.501,Z 165.362,A -85,B 0,C 180,E1 -3724.53,E2 -3724.53} C_VEL
LIN {X 0,Y 545.498,Z 162.465,A -85,B 0,C 180,E1 -3725.74,E2 -3725.74} C_VEL
LIN {X 0,Y 545.059,Z 159.594,A -85,B 0,C 180,E1 -3727.082,E2 -3727.082} C_VEL
LIN {X 0,Y 545.059,Z 159.596,A -85,B 0,C 180,E1 -3730.14,E2 -3730.14} C_VEL
LIN {X 0,Y 545.076,Z 159.587,A -85,B 0,C 180,E1 -3733.104,E2 -3733.104} C_VEL
LIN {X 0,Y 545.042,Z 159.59,A -85,B 0,C 180,E1 -3736.223,E2 -3736.223} C_VEL
LIN {X 0,Y 545.065,Z 159.591,A -85,B 0,C 180,E1 -3738.884,E2 -3738.884} C_VEL
LIN {X 0,Y 545.062,Z 159.589,A -85,B 0,C 180,E1 -3740.817,E2 -3740.817} C_VEL
LIN {X 0,Y 545.041,Z 159.597,A -85,B 0,C 180,E1 -3743.62,E2 -3743.62} C_VEL
LIN {X 0,Y 545.058,Z 159.588,A -85,B 0,C 180,E1 -3746.328,E2 -3746.328} C_VEL
LIN {X 0,Y 545.048,Z 159.594,A -85,B 0,C 180,E1 -3748.951,E2 -3748.951} C_VEL
LIN {X 0,Y 545.079,Z 159.587,A -85,B 0,C 180,E1 -3751.506,E2 -3751.506} C_VEL
LIN {X 0,Y 545.067,Z 159.587,A -85,B 0,C 180,E1 -3754.49,E2 -3754.49} C_VEL
LIN {X 0,Y 545.054,Z 159.593,A -85,B 0,C 180,E1 -3757.243,E2 -3757.243} C_VEL
LIN {X 0,Y 545.093,Z 159.588,A -85,B 0,C 180,E1 -3760.414,E2 -3760.414} C_VEL
LIN {X 0,Y 545.121,Z 159.582,A -85,B 0,C 180,E1 -3762.751,E2 -3762.751} C_VEL
LIN {X 0,Y 545.064,Z 159.591,A -85,B 0,C 180,E1 -3765.819,E2 -3765.819} C_VEL
LIN {X 0,Y 545.148,Z 159.583,A -85,B 0,C 180,E1 -3768.85,E2 -3768.85} C_VEL
LIN {X 0,Y 545.115,Z 159.582,A -85,B 0,C 180,E1 -3771.847,E2 -3771.847} C_VEL
LIN {X 0,Y 545.166,Z 159.58,A -85,B 0,C 180,E1 -3774.081,E2 -3774.081} C_VEL
LIN {X 0,Y 545.149,Z 159.581,A -85,B 0,C 180,E1 -3777.044,E2 -3777.044} C_VEL
LIN {X 0,Y 545.163,Z 159.576,A -85,B 0,C 180,E1 -3780,E2 -3780} C_VEL
LIN {X 0,Y 545.157,Z 159.576,A -85,B 0,C 180,E1 -3782.956,E2 -3782.956} C_VEL
LIN {X 0,Y 545.161,Z 159.58,A -85,B 0,C 180,E1 -3785.92,E2 -3785.92} C_VEL
LIN {X 0,Y 545.102,Z 159.587,A -85,B 0,C 180,E1 -3788.901,E2 -3788.901} C_VEL
LIN {X 0,Y 545.105,Z 159.584,A -85,B 0,C 180,E1 -3791.905,E2 -3791.905} C_VEL
LIN {X 0,Y 545.059,Z 159.588,A -85,B 0,C 180,E1 -3794.945,E2 -3794.945} C_VEL
LIN {X 0,Y 545.116,Z 159.586,A -85,B 0,C 180,E1 -3797.447,E2 -3797.447} C_VEL
LIN {X 0,Y 545.076,Z 159.587,A -85,B 0,C 180,E1 -3800.373,E2 -3800.373} C_VEL
LIN {X 0,Y 545.067,Z 159.588,A -85,B 0,C 180,E1 -3803.56,E2 -3803.56} C_VEL
LIN {X 0,Y 545.064,Z 159.592,A -85,B 0,C 180,E1 -3806.002,E2 -3806.002} C_VEL
LIN {X 0,Y 545.071,Z 159.587,A -85,B 0,C 180,E1 -3808.751,E2 -3808.751} C_VEL
LIN {X 0,Y 545.057,Z 159.588,A -85,B 0,C 180,E1 -3811.684,E2 -3811.684} C_VEL
LIN {X 0,Y 545.06,Z 159.592,A -85,B 0,C 180,E1 -3814.565,E2 -3814.565} C_VEL
LIN {X 0,Y 545.041,Z 159.591,A -85,B 0,C 180,E1 -3817.037,E2 -3817.037} C_VEL
LIN {X 0,Y 544.335,Z 159.683,A -85,B 0,C 180,E1 -3817.653,E2 -3817.653} C_VEL
LIN {X 0,Y 541.472,Z 160.037,A -85,B 0,C 180,E1 -3818.654,E2 -3818.654} C_VEL
LIN {X 0,Y 539.088,Z 160.336,A -85,B 0,C 180,E1 -3819.46,E2 -3819.46} C_VEL
LIN {X 0,Y 538.081,Z 160.458,A -85,B 0,C 180,E1 -3820.082,E2 -3820.082} C_VEL
LIN {X 0,Y 538.006,Z 160.466,A -85,B 0,C 180,E1 -3820.293,E2 -3820.293} C_VEL
LIN {X 0,Y 538.012,Z 160.469,A -85,B 0,C 180,E1 -3822.99,E2 -3822.99} C_VEL
LIN {X 0,Y 538.009,Z 160.47,A -85,B 0,C 180,E1 -3825.928,E2 -3825.928} C_VEL
LIN {X 0,Y 538.038,Z 160.467,A -85,B 0,C 180,E1 -3829.226,E2 -3829.226} C_VEL
LIN {X 0,Y 537.948,Z 160.475,A -85,B 0,C 180,E1 -3832.121,E2 -3832.121} C_VEL
LIN {X 0,Y 537.916,Z 161.075,A -85,B 0,C 180,E1 -3833.061,E2 -3833.061} C_VEL
LIN {X 0,Y 537.904,Z 165.341,A -85,B 0,C 180,E1 -3835.821,E2 -3835.821} C_VEL
LIN {X 0,Y 537.864,Z 169.552,A -85,B 0,C 180,E1 -3838.491,E2 -3838.491} C_VEL
LIN {X 0,Y 537.828,Z 173.763,A -85,B 0,C 180,E1 -3841.107,E2 -3841.107} C_VEL
LIN {X 0,Y 537.728,Z 177.893,A -85,B 0,C 180,E1 -3843.618,E2 -3843.618} C_VEL
LIN {X 0,Y 537.715,Z 182.218,A -85,B 0,C 180,E1 -3846.194,E2 -3846.194} C_VEL
LIN {X 0,Y 537.646,Z 186.186,A -85,B 0,C 180,E1 -3848.531,E2 -3848.531} C_VEL
LIN {X 0,Y 537.612,Z 190.377,A -85,B 0,C 180,E1 -3850.925,E2 -3850.925} C_VEL
LIN {X 0,Y 537.573,Z 194.456,A -85,B 0,C 180,E1 -3853.285,E2 -3853.285} C_VEL
LIN {X 0,Y 537.545,Z 196.963,A -85,B 0,C 180,E1 -3854.721,E2 -3854.721} C_VEL
LIN {X 0,Y 539.244,Z 207.672,A -85,B 0,C 180,E1 -3855.034,E2 -3855.034} C_VEL
LIN {X 0,Y 538.997,Z 220.616,A -85,B 0,C 180,E1 -3855.483,E2 -3855.483} C_VEL
LIN {X 0,Y 538.756,Z 232.223,A -85,B 0,C 180,E1 -3856.035,E2 -3856.035} C_VEL
LIN {X 0,Y 538.483,Z 243.124,A -85,B 0,C 180,E1 -3856.701,E2 -3856.701} C_VEL
LIN {X 0,Y 538.334,Z 254.217,A -85,B 0,C 180,E1 -3857.561,E2 -3857.561} C_VEL
LIN {X 0,Y 538.08,Z 264.532,A -85,B 0,C 180,E1 -3858.56,E2 -3858.56} C_VEL
LIN {X 0,Y 537.941,Z 273.61,A -85,B 0,C 180,E1 -3859.652,E2 -3859.652} C_VEL
LIN {X 0,Y 537.78,Z 281.175,A -85,B 0,C 180,E1 -3860.788,E2 -3860.788} C_VEL
LIN {X 0,Y 537.663,Z 288.15,A -85,B 0,C 180,E1 -3862.111,E2 -3862.111} C_VEL
LIN {X 0,Y 537.621,Z 292.763,A -85,B 0,C 180,E1 -3863.243,E2 -3863.243} C_VEL
LIN {X 0,Y 537.558,Z 295.21,A -85,B 0,C 180,E1 -3863.996,E2 -3863.996} C_VEL
LIN {X 0,Y 537.539,Z 297.198,A -85,B 0,C 180,E1 -3864.749,E2 -3864.749} C_VEL
LIN {X 0,Y 537.501,Z 298.773,A -85,B 0,C 180,E1 -3865.5,E2 -3865.5} C_VEL
LIN {X 0,Y 537.563,Z 299.937,A -85,B 0,C 180,E1 -3866.252,E2 -3866.252} C_VEL
LIN {X 0,Y 537.546,Z 300.665,A -85,B 0,C 180,E1 -3867.002,E2 -3867.002} C_VEL
LIN {X 0,Y 537.451,Z 300.978,A -85,B 0,C 180,E1 -3868.501,E2 -3868.501} C_VEL
LIN {X 0,Y 537.442,Z 300.559,A -85,B 0,C 180,E1 -3869.25,E2 -3869.25} C_VEL
LIN {X 0,Y 537.446,Z 299.709,A -85,B 0,C 180,E1 -3869.999,E2 -3869.999} C_VEL
LIN {X 0,Y 537.479,Z 296.827,A -85,B 0,C 180,E1 -3871.498,E2 -3871.498} C_VEL
LIN {X 0,Y 537.579,Z 293.531,A -85,B 0,C 180,E1 -3872.622,E2 -3872.622} C_VEL
LIN {X 0,Y 537.646,Z 289.178,A -85,B 0,C 180,E1 -3873.747,E2 -3873.747} C_VEL
LIN {X 0,Y 537.805,Z 283.643,A -85,B 0,C 180,E1 -3874.872,E2 -3874.872} C_VEL
LIN {X 0,Y 537.843,Z 276.745,A -85,B 0,C 180,E1 -3875.999,E2 -3875.999} C_VEL
LIN {X 0,Y 538.01,Z 268.103,A -85,B 0,C 180,E1 -3877.127,E2 -3877.127} C_VEL
LIN {X 0,Y 538.273,Z 259.248,A -85,B 0,C 180,E1 -3878.067,E2 -3878.067} C_VEL
LIN {X 0,Y 538.443,Z 249.53,A -85,B 0,C 180,E1 -3878.916,E2 -3878.916} C_VEL
LIN {X 0,Y 538.582,Z 238.84,A -85,B 0,C 180,E1 -3879.671,E2 -3879.671} C_VEL
LIN {X 0,Y 538.879,Z 226.84,A -85,B 0,C 180,E1 -3880.329,E2 -3880.329} C_VEL
LIN {X 0,Y 539.114,Z 214.553,A -85,B 0,C 180,E1 -3880.838,E2 -3880.838} C_VEL
LIN {X 0,Y 539.051,Z 205.549,A -85,B 0,C 180,E1 -3881.117,E2 -3881.117} C_VEL
LIN {X 0,Y 537.591,Z 196.915,A -85,B 0,C 180,E1 -3881.369,E2 -3881.369} C_VEL
LIN {X 0,Y 537.653,Z 191.081,A -85,B 0,C 180,E1 -3884.691,E2 -3884.691} C_VEL
LIN {X 0,Y 537.657,Z 186.289,A -85,B 0,C 180,E1 -3887.495,E2 -3887.495} C_VEL
LIN {X 0,Y 537.721,Z 182.262,A -85,B 0,C 180,E1 -3889.864,E2 -3889.864} C_VEL
LIN {X 0,Y 537.767,Z 178.217,A -85,B 0,C 180,E1 -3892.269,E2 -3892.269} C_VEL
LIN {X 0,Y 537.797,Z 174.173,A -85,B 0,C 180,E1 -3894.717,E2 -3894.717} C_VEL
LIN {X 0,Y 537.833,Z 169.971,A -85,B 0,C 180,E1 -3897.305,E2 -3897.305} C_VEL
LIN {X 0,Y 537.888,Z 166.034,A -85,B 0,C 180,E1 -3899.766,E2 -3899.766} C_VEL
LIN {X 0,Y 537.895,Z 161.899,A -85,B 0,C 180,E1 -3902.388,E2 -3902.388} C_VEL
LIN {X 0,Y 537.897,Z 160.506,A -85,B 0,C 180,E1 -3903.279,E2 -3903.279} C_VEL
LIN {X 0,Y 537.977,Z 160.47,A -85,B 0,C 180,E1 -3905.908,E2 -3905.908} C_VEL
LIN {X 0,Y 537.997,Z 160.471,A -85,B 0,C 180,E1 -3908.828,E2 -3908.828} C_VEL
LIN {X 0,Y 538.026,Z 160.469,A -85,B 0,C 180,E1 -3911.769,E2 -3911.769} C_VEL
LIN {X 0,Y 538.014,Z 160.466,A -85,B 0,C 180,E1 -3914.857,E2 -3914.857} C_VEL
LIN {X 0,Y 538.032,Z 160.462,A -85,B 0,C 180,E1 -3918.116,E2 -3918.116} C_VEL
LIN {X 0,Y 538.036,Z 160.465,A -85,B 0,C 180,E1 -3920.409,E2 -3920.409} C_VEL
LIN {X 0,Y 538,Z 160.468,A -85,B 0,C 180,E1 -3923.065,E2 -3923.065} C_VEL
LIN {X 0,Y 538.001,Z 160.472,A -85,B 0,C 180,E1 -3925.825,E2 -3925.825} C_VEL
LIN {X 0,Y 537.996,Z 160.468,A -85,B 0,C 180,E1 -3928.497,E2 -3928.497} C_VEL
LIN {X 0,Y 538.029,Z 160.47,A -85,B 0,C 180,E1 -3931.098,E2 -3931.098} C_VEL
LIN {X 0,Y 538.037,Z 160.462,A -85,B 0,C 180,E1 -3933.633,E2 -3933.633} C_VEL
LIN {X 0,Y 538.044,Z 160.464,A -85,B 0,C 180,E1 -3936.113,E2 -3936.113} C_VEL
LIN {X 0,Y 538.007,Z 160.467,A -85,B 0,C 180,E1 -3939.347,E2 -3939.347} C_VEL
LIN {X 0,Y 538.036,Z 160.463,A -85,B 0,C 180,E1 -3942.516,E2 -3942.516} C_VEL
LIN {X 0,Y 538.031,Z 160.465,A -85,B 0,C 180,E1 -3945.63,E2 -3945.63} C_VEL
LIN {X 0,Y 538.115,Z 160.457,A -85,B 0,C 180,E1 -3948.702,E2 -3948.702} C_VEL
LIN {X 0,Y 538.076,Z 160.46,A -85,B 0,C 180,E1 -3951.739,E2 -3951.739} C_VEL
LIN {X 0,Y 538.13,Z 160.455,A -85,B 0,C 180,E1 -3954.003,E2 -3954.003} C_VEL
LIN {X 0,Y 538.109,Z 160.457,A -85,B 0,C 180,E1 -3957.005,E2 -3957.005} C_VEL
LIN {X 0,Y 538.125,Z 160.452,A -85,B 0,C 180,E1 -3960,E2 -3960} C_VEL
LIN {X 0,Y 538.116,Z 160.455,A -85,B 0,C 180,E1 -3962.994,E2 -3962.994} C_VEL
LIN {X 0,Y 538.13,Z 160.457,A -85,B 0,C 180,E1 -3965.997,E2 -3965.997} C_VEL
LIN {X 0,Y 538.076,Z 160.458,A -85,B 0,C 180,E1 -3968.26,E2 -3968.26} C_VEL
LIN {X 0,Y 538.068,Z 160.461,A -85,B 0,C 180,E1 -3971.611,E2 -3971.611} C_VEL
LIN {X 0,Y 538.019,Z 160.471,A -85,B 0,C 180,E1 -3974.858,E2 -3974.858} C_VEL
LIN {X 0,Y 538.021,Z 160.465,A -85,B 0,C 180,E1 -3977.542,E2 -3977.542} C_VEL
LIN {X 0,Y 538.008,Z 160.467,A -85,B 0,C 180,E1 -3980.653,E2 -3980.653} C_VEL
LIN {X 0,Y 538.043,Z 160.463,A -85,B 0,C 180,E1 -3983.887,E2 -3983.887} C_VEL
LIN {X 0,Y 538.035,Z 160.463,A -85,B 0,C 180,E1 -3986.367,E2 -3986.367} C_VEL
LIN {X 0,Y 538.044,Z 160.465,A -85,B 0,C 180,E1 -3988.944,E2 -3988.944} C_VEL
LIN {X 0,Y 537.997,Z 160.471,A -85,B 0,C 180,E1 -3991.892,E2 -3991.892} C_VEL
LIN {X 0,Y 537.997,Z 160.468,A -85,B 0,C 180,E1 -3994.622,E2 -3994.622} C_VEL
LIN {X 0,Y 537.981,Z 160.474,A -85,B 0,C 180,E1 -3997.173,E2 -3997.173} C_VEL
LIN {X 0,Y 538.031,Z 160.464,A -85,B 0,C 180,E1 -3999.796,E2 -3999.796} C_VEL
LIN {X 0,Y 538.003,Z 160.471,A -85,B 0,C 180,E1 -4002.788,E2 -4002.788} C_VEL
LIN {X 0,Y 538.009,Z 160.47,A -85,B 0,C 180,E1 -4005.928,E2 -4005.928} C_VEL
LIN {X 0,Y 538.034,Z 160.468,A -85,B 0,C 180,E1 -4009.227,E2 -4009.227} C_VEL
LIN {X 0,Y 537.974,Z 160.474,A -85,B 0,C 180,E1 -4012.125,E2 -4012.125} C_VEL
LIN {X 0,Y 538.014,Z 160.53,A -85,B 0,C 180,E1 -4012.983,E2 -4012.983} C_VEL
LIN {X 0,Y 538.527,Z 165.124,A -85,B 0,C 180,E1 -4014.959,E2 -4014.959} C_VEL
LIN {X 0,Y 538.392,Z 172.772,A -85,B 0,C 180,E1 -4018.048,E2 -4018.048} C_VEL
LIN {X 0,Y 538.241,Z 180.693,A -85,B 0,C 180,E1 -4021.113,E2 -4021.113} C_VEL
LIN {X 0,Y 538.103,Z 189.661,A -85,B 0,C 180,E1 -4024.471,E2 -4024.471} C_VEL
LIN {X 0,Y 537.943,Z 197.51,A -85,B 0,C 180,E1 -4027.333,E2 -4027.333} C_VEL
LIN {X 0,Y 537.834,Z 205.507,A -85,B 0,C 180,E1 -4030.194,E2 -4030.194} C_VEL
LIN {X 0,Y 537.738,Z 213.266,A -85,B 0,C 180,E1 -4032.927,E2 -4032.927} C_VEL
LIN {X 0,Y 537.708,Z 222.27,A -85,B 0,C 180,E1 -4036.009,E2 -4036.009} C_VEL
LIN {X 0,Y 537.652,Z 224.179,A -85,B 0,C 180,E1 -4036.658,E2 -4036.658} C_VEL
LIN {X 0,Y 539.206,Z 234.988,A -85,B 0,C 180,E1 -4036.936,E2 -4036.936} C_VEL
LIN {X 0,Y 539.004,Z 247.497,A -85,B 0,C 180,E1 -4037.338,E2 -4037.338} C_VEL
LIN {X 0,Y 538.805,Z 259.14,A -85,B 0,C 180,E1 -4037.86,E2 -4037.86} C_VEL
LIN {X 0,Y 538.557,Z 269.917,A -85,B 0,C 180,E1 -4038.483,E2 -4038.483} C_VEL
LIN {X 0,Y 538.356,Z 280.878,A -85,B 0,C 180,E1 -4039.28,E2 -4039.28} C_VEL
LIN {X 0,Y 538.124,Z 291.362,A -85,B 0,C 180,E1 -4040.226,E2 -4040.226} C_VEL
LIN {X 0,Y 537.965,Z 299.847,A -85,B 0,C 180,E1 -4041.171,E2 -4041.171} C_VEL
LIN {X 0,Y 537.796,Z 308.126,A -85,B 0,C 180,E1 -4042.303,E2 -4042.303} C_VEL
LIN {X 0,Y 537.654,Z 314.812,A -85,B 0,C 180,E1 -4043.436,E2 -4043.436} C_VEL
LIN {X 0,Y 537.676,Z 319.315,A -85,B 0,C 180,E1 -4044.375,E2 -4044.375} C_VEL
LIN {X 0,Y 537.556,Z 323.647,A -85,B 0,C 180,E1 -4045.502,E2 -4045.502} C_VEL
LIN {X 0,Y 537.591,Z 325.943,A -85,B 0,C 180,E1 -4046.253,E2 -4046.253} C_VEL
LIN {X 0,Y 537.551,Z 327.801,A -85,B 0,C 180,E1 -4047.003,E2 -4047.003} C_VEL
LIN {X 0,Y 537.451,Z 330.181,A -85,B 0,C 180,E1 -4048.502,E2 -4048.502} C_VEL
LIN {X 0,Y 537.442,Z 331,A -85,B 0,C 180,E1 -4050.001,E2 -4050.001} C_VEL
LIN {X 0,Y 537.451,Z 330.182,A -85,B 0,C 180,E1 -4051.499,E2 -4051.499} C_VEL
LIN {X 0,Y 537.49,Z 329.193,A -85,B 0,C 180,E1 -4052.248,E2 -4052.248} C_VEL
LIN {X 0,Y 537.551,Z 327.803,A -85,B 0,C 180,E1 -4052.998,E2 -4052.998} C_VEL
LIN {X 0,Y 537.603,Z 324.871,A -85,B 0,C 180,E1 -4054.123,E2 -4054.123} C_VEL
LIN {X 0,Y 537.587,Z 320.899,A -85,B 0,C 180,E1 -4055.251,E2 -4055.251} C_VEL
LIN {X 0,Y 537.64,Z 316.053,A -85,B 0,C 180,E1 -4056.326,E2 -4056.326} C_VEL
LIN {X 0,Y 537.772,Z 309.356,A -85,B 0,C 180,E1 -4057.509,E2 -4057.509} C_VEL
LIN {X 0,Y 537.953,Z 301.33,A -85,B 0,C 180,E1 -4058.641,E2 -4058.641} C_VEL
LIN {X 0,Y 538.089,Z 293.151,A -85,B 0,C 180,E1 -4059.586,E2 -4059.586} C_VEL
LIN {X 0,Y 538.362,Z 283.179,A -85,B 0,C 180,E1 -4060.53,E2 -4060.53} C_VEL
LIN {X 0,Y 538.497,Z 273.341,A -85,B 0,C 180,E1 -4061.289,E2 -4061.289} C_VEL
LIN {X 0,Y 538.713,Z 262.326,A -85,B 0,C 180,E1 -4061.97,E2 -4061.97} C_VEL
LIN {X 0,Y 538.956,Z 249.796,A -85,B 0,C 180,E1 -4062.568,E2 -4062.568} C_VEL
LIN {X 0,Y 539.187,Z 236.767,A -85,B 0,C 180,E1 -4063.017,E2 -4063.017} C_VEL
LIN {X 0,Y 538.933,Z 232.182,A -85,B 0,C 180,E1 -4063.143,E2 -4063.143} C_VEL
LIN {X 0,Y 537.642,Z 224.173,A -85,B 0,C 180,E1 -4063.344,E2 -4063.344} C_VEL
LIN {X 0,Y 537.74,Z 216.668,A -85,B 0,C 180,E1 -4065.929,E2 -4065.929} C_VEL
LIN {X 0,Y 537.79,Z 208.738,A -85,B 0,C 180,E1 -4068.673,E2 -4068.673} C_VEL
LIN {X 0,Y 537.895,Z 200.852,A -85,B 0,C 180,E1 -4071.458,E2 -4071.458} C_VEL
LIN {X 0,Y 538.008,Z 193,A -85,B 0,C 180,E1 -4074.297,E2 -4074.297} C_VEL
LIN {X 0,Y 538.12,Z 185.176,A -85,B 0,C 180,E1 -4077.199,E2 -4077.199} C_VEL
LIN {X 0,Y 538.28,Z 178.504,A -85,B 0,C 180,E1 -4079.743,E2 -4079.743} C_VEL
LIN {X 0,Y 538.431,Z 170.785,A -85,B 0,C 180,E1 -4082.797,E2 -4082.797} C_VEL
LIN {X 0,Y 538.55,Z 164.265,A -85,B 0,C 180,E1 -4085.499,E2 -4085.499} C_VEL
LIN {X 0,Y 538.031,Z 160.47,A -85,B 0,C 180,E1 -4087.203,E2 -4087.203} C_VEL
LIN {X 0,Y 538.013,Z 160.472,A -85,B 0,C 180,E1 -4089.795,E2 -4089.795} C_VEL
LIN {X 0,Y 538.012,Z 160.466,A -85,B 0,C 180,E1 -4092.783,E2 -4092.783} C_VEL
LIN {X 0,Y 538.018,Z 160.47,A -85,B 0,C 180,E1 -4095.139,E2 -4095.139} C_VEL
LIN {X 0,Y 538.014,Z 160.468,A -85,B 0,C 180,E1 -4098.225,E2 -4098.225} C_VEL
LIN {X 0,Y 537.994,Z 160.469,A -85,B 0,C 180,E1 -4101.168,E2 -4101.168} C_VEL
LIN {X 0,Y 538.011,Z 160.467,A -85,B 0,C 180,E1 -4104.081,E2 -4104.081} C_VEL
LIN {X 0,Y 538.015,Z 160.468,A -85,B 0,C 180,E1 -4106.726,E2 -4106.726} C_VEL
LIN {X 0,Y 538.015,Z 160.466,A -85,B 0,C 180,E1 -4109.552,E2 -4109.552} C_VEL
LIN {X 0,Y 538.021,Z 160.469,A -85,B 0,C 180,E1 -4111.949,E2 -4111.949} C_VEL
LIN {X 0,Y 538.044,Z 160.462,A -85,B 0,C 180,E1 -4114.466,E2 -4114.466} C_VEL
LIN {X 0,Y 538.036,Z 160.467,A -85,B 0,C 180,E1 -4116.929,E2 -4116.929} C_VEL
LIN {X 0,Y 538.051,Z 160.463,A -85,B 0,C 180,E1 -4120.147,E2 -4120.147} C_VEL
LIN {X 0,Y 538.028,Z 160.465,A -85,B 0,C 180,E1 -4123.299,E2 -4123.299} C_VEL
LIN {X 0,Y 538.033,Z 160.468,A -85,B 0,C 180,E1 -4125.63,E2 -4125.63} C_VEL
LIN {X 0,Y 538.092,Z 160.46,A -85,B 0,C 180,E1 -4128.702,E2 -4128.702} C_VEL
LIN {X 0,Y 538.07,Z 160.459,A -85,B 0,C 180,E1 -4131.739,E2 -4131.739} C_VEL
LIN {X 0,Y 538.14,Z 160.456,A -85,B 0,C 180,E1 -4134.003,E2 -4134.003} C_VEL
LIN {X 0,Y 538.115,Z 160.457,A -85,B 0,C 180,E1 -4137.006,E2 -4137.006} C_VEL
LIN {X 0,Y 538.134,Z 160.451,A -85,B 0,C 180,E1 -4140,E2 -4140} C_VEL
LIN {X 0,Y 538.123,Z 160.452,A -85,B 0,C 180,E1 -4142.995,E2 -4142.995} C_VEL
LIN {X 0,Y 538.111,Z 160.457,A -85,B 0,C 180,E1 -4145.998,E2 -4145.998} C_VEL
LIN {X 0,Y 538.051,Z 160.465,A -85,B 0,C 180,E1 -4149.018,E2 -4149.018} C_VEL
LIN {X 0,Y 538.053,Z 160.463,A -85,B 0,C 180,E1 -4152.063,E2 -4152.063} C_VEL
LIN {X 0,Y 538.02,Z 160.465,A -85,B 0,C 180,E1 -4155.145,E2 -4155.145} C_VEL
LIN {X 0,Y 538.066,Z 160.465,A -85,B 0,C 180,E1 -4157.553,E2 -4157.553} C_VEL
LIN {X 0,Y 538.019,Z 160.469,A -85,B 0,C 180,E1 -4160.652,E2 -4160.652} C_VEL
LIN {X 0,Y 537.999,Z 160.471,A -85,B 0,C 180,E1 -4163.889,E2 -4163.889} C_VEL
LIN {X 0,Y 538.025,Z 160.466,A -85,B 0,C 180,E1 -4166.368,E2 -4166.368} C_VEL
LIN {X 0,Y 538.034,Z 160.465,A -85,B 0,C 180,E1 -4168.94,E2 -4168.94} C_VEL
LIN {X 0,Y 538.008,Z 160.466,A -85,B 0,C 180,E1 -4171.892,E2 -4171.892} C_VEL
LIN {X 0,Y 538.009,Z 160.47,A -85,B 0,C 180,E1 -4174.622,E2 -4174.622} C_VEL
LIN {X 0,Y 537.986,Z 160.471,A -85,B 0,C 180,E1 -4177.172,E2 -4177.172} C_VEL
LIN {X 0,Y 538.006,Z 160.466,A -85,B 0,C 180,E1 -4180.293,E2 -4180.293} C_VEL
LIN {X 0,Y 537.358,Z 160.552,A -85,B 0,C 180,E1 -4180.918,E2 -4180.918} C_VEL
LIN {X 0,Y 534.507,Z 160.904,A -85,B 0,C 180,E1 -4181.933,E2 -4181.933} C_VEL
LIN {X 0,Y 532.082,Z 161.211,A -85,B 0,C 180,E1 -4182.75,E2 -4182.75} C_VEL
LIN {X 0,Y 531.035,Z 161.335,A -85,B 0,C 180,E1 -4183.381,E2 -4183.381} C_VEL
LIN {X 0,Y 530.948,Z 161.345,A -85,B 0,C 180,E1 -4183.595,E2 -4183.595} C_VEL
LIN {X 0,Y 530.943,Z 161.349,A -85,B 0,C 180,E1 -4186.506,E2 -4186.506} C_VEL
LIN {X 0,Y 530.975,Z 161.345,A -85,B 0,C 180,E1 -4188.978,E2 -4188.978} C_VEL
LIN {X 0,Y 530.932,Z 161.351,A -85,B 0,C 180,E1 -4191.53,E2 -4191.53} C_VEL
LIN {X 0,Y 530.862,Z 161.361,A -85,B 0,C 180,E1 -4192.593,E2 -4192.593} C_VEL
LIN {X 0,Y 530.877,Z 165.376,A -85,B 0,C 180,E1 -4195.304,E2 -4195.304} C_VEL
LIN {X 0,Y 530.834,Z 169.604,A -85,B 0,C 180,E1 -4198.025,E2 -4198.025} C_VEL
LIN {X 0,Y 530.779,Z 174.193,A -85,B 0,C 180,E1 -4200.916,E2 -4200.916} C_VEL
LIN {X 0,Y 530.673,Z 179.342,A -85,B 0,C 180,E1 -4204.086,E2 -4204.086} C_VEL
LIN {X 0,Y 530.621,Z 183.51,A -85,B 0,C 180,E1 -4206.589,E2 -4206.589} C_VEL
LIN {X 0,Y 530.568,Z 189.06,A -85,B 0,C 180,E1 -4209.856,E2 -4209.856} C_VEL
LIN {X 0,Y 530.506,Z 194.612,A -85,B 0,C 180,E1 -4213.056,E2 -4213.056} C_VEL
LIN {X 0,Y 530.491,Z 197.25,A -85,B 0,C 180,E1 -4214.559,E2 -4214.559} C_VEL
LIN {X 0,Y 532.316,Z 208.262,A -85,B 0,C 180,E1 -4214.873,E2 -4214.873} C_VEL
LIN {X 0,Y 532.081,Z 220.694,A -85,B 0,C 180,E1 -4215.312,E2 -4215.312} C_VEL
LIN {X 0,Y 531.835,Z 231.932,A -85,B 0,C 180,E1 -4215.85,E2 -4215.85} C_VEL
LIN {X 0,Y 531.533,Z 242.928,A -85,B 0,C 180,E1 -4216.524,E2 -4216.524} C_VEL
LIN {X 0,Y 531.356,Z 254.119,A -85,B 0,C 180,E1 -4217.395,E2 -4217.395} C_VEL
LIN {X 0,Y 531.134,Z 263.382,A -85,B 0,C 180,E1 -4218.288,E2 -4218.288} C_VEL
LIN {X 0,Y 530.942,Z 272.14,A -85,B 0,C 180,E1 -4219.321,E2 -4219.321} C_VEL
LIN {X 0,Y 530.716,Z 280.085,A -85,B 0,C 180,E1 -4220.472,E2 -4220.472} C_VEL
LIN {X 0,Y 530.608,Z 286.419,A -85,B 0,C 180,E1 -4221.622,E2 -4221.622} C_VEL
LIN {X 0,Y 530.567,Z 291.442,A -85,B 0,C 180,E1 -4222.771,E2 -4222.771} C_VEL
LIN {X 0,Y 530.471,Z 295.335,A -85,B 0,C 180,E1 -4223.916,E2 -4223.916} C_VEL
LIN {X 0,Y 530.463,Z 297.334,A -85,B 0,C 180,E1 -4224.679,E2 -4224.679} C_VEL
LIN {X 0,Y 530.406,Z 298.922,A -85,B 0,C 180,E1 -4225.44,E2 -4225.44} C_VEL
LIN {X 0,Y 530.482,Z 300.102,A -85,B 0,C 180,E1 -4226.202,E2 -4226.202} C_VEL
LIN {X 0,Y 530.41,Z 301.203,A -85,B 0,C 180,E1 -4227.722,E2 -4227.722} C_VEL
LIN {X 0,Y 530.346,Z 300.777,A -85,B 0,C 180,E1 -4229.24,E2 -4229.24} C_VEL
LIN {X 0,Y 530.35,Z 299.946,A -85,B 0,C 180,E1 -4229.999,E2 -4229.999} C_VEL
LIN {X 0,Y 530.39,Z 297.085,A -85,B 0,C 180,E1 -4231.518,E2 -4231.518} C_VEL
LIN {X 0,Y 530.498,Z 293.813,A -85,B 0,C 180,E1 -4232.657,E2 -4232.657} C_VEL
LIN {X 0,Y 530.57,Z 289.486,A -85,B 0,C 180,E1 -4233.797,E2 -4233.797} C_VEL
LIN {X 0,Y 530.747,Z 283.978,A -85,B 0,C 180,E1 -4234.937,E2 -4234.937} C_VEL
LIN {X 0,Y 530.806,Z 277.118,A -85,B 0,C 180,E1 -4236.079,E2 -4236.079} C_VEL
LIN {X 0,Y 530.985,Z 268.523,A -85,B 0,C 180,E1 -4237.222,E2 -4237.222} C_VEL
LIN {X 0,Y 531.261,Z 259.713,A -85,B 0,C 180,E1 -4238.175,E2 -4238.175} C_VEL
LIN {X 0,Y 531.506,Z 248.869,A -85,B 0,C 180,E1 -4239.129,E2 -4239.129} C_VEL
LIN {X 0,Y 531.72,Z 237.895,A -85,B 0,C 180,E1 -4239.893,E2 -4239.893} C_VEL
LIN {X 0,Y 531.995,Z 225.607,A -85,B 0,C 180,E1 -4240.561,E2 -4240.561} C_VEL
LIN {X 0,Y 532.23,Z 213.395,A -85,B 0,C 180,E1 -4241.056,E2 -4241.056} C_VEL
LIN {X 0,Y 532.15,Z 206.582,A -85,B 0,C 180,E1 -4241.267,E2 -4241.267} C_VEL
LIN {X 0,Y 530.515,Z 197.122,A -85,B 0,C 180,E1 -4241.547,E2 -4241.547} C_VEL
LIN {X 0,Y 530.586,Z 191.537,A -85,B 0,C 180,E1 -4244.772,E2 -4244.772} C_VEL
LIN {X 0,Y 530.593,Z 186.466,A -85,B 0,C 180,E1 -4247.735,E2 -4247.735} C_VEL
LIN {X 0,Y 530.663,Z 182.425,A -85,B 0,C 180,E1 -4250.139,E2 -4250.139} C_VEL
LIN {X 0,Y 530.68,Z 178.375,A -85,B 0,C 180,E1 -4252.583,E2 -4252.583} C_VEL
LIN {X 0,Y 530.722,Z 174.319,A -85,B 0,C 180,E1 -4255.069,E2 -4255.069} C_VEL
LIN {X 0,Y 530.781,Z 170.247,A -85,B 0,C 180,E1 -4257.606,E2 -4257.606} C_VEL
LIN {X 0,Y 530.868,Z 165.482,A -85,B 0,C 180,E1 -4260.625,E2 -4260.625} C_VEL
LIN {X 0,Y 530.848,Z 161.999,A -85,B 0,C 180,E1 -4262.872,E2 -4262.872} C_VEL
LIN {X 0,Y 530.875,Z 161.361,A -85,B 0,C 180,E1 -4263.484,E2 -4263.484} C_VEL
LIN {X 0,Y 530.937,Z 161.348,A -85,B 0,C 180,E1 -4265.618,E2 -4265.618} C_VEL
LIN {X 0,Y 530.95,Z 161.35,A -85,B 0,C 180,E1 -4268.651,E2 -4268.651} C_VEL
LIN {X 0,Y 530.985,Z 161.342,A -85,B 0,C 180,E1 -4271.432,E2 -4271.432} C_VEL
LIN {X 0,Y 530.97,Z 161.343,A -85,B 0,C 180,E1 -4274.544,E2 -4274.544} C_VEL
LIN {X 0,Y 530.977,Z 161.341,A -85,B 0,C 180,E1 -4277.83,E2 -4277.83} C_VEL
LIN {X 0,Y 530.982,Z 161.345,A -85,B 0,C 180,E1 -4280.556,E2 -4280.556} C_VEL
LIN {X 0,Y 530.932,Z 161.348,A -85,B 0,C 180,E1 -4283.439,E2 -4283.439} C_VEL
LIN {X 0,Y 530.972,Z 161.344,A -85,B 0,C 180,E1 -4286.492,E2 -4286.492} C_VEL
LIN {X 0,Y 530.953,Z 161.35,A -85,B 0,C 180,E1 -4289.351,E2 -4289.351} C_VEL
LIN {X 0,Y 530.975,Z 161.344,A -85,B 0,C 180,E1 -4291.543,E2 -4291.543} C_VEL
LIN {X 0,Y 530.995,Z 161.34,A -85,B 0,C 180,E1 -4294.15,E2 -4294.15} C_VEL
LIN {X 0,Y 530.979,Z 161.345,A -85,B 0,C 180,E1 -4296.604,E2 -4296.604} C_VEL
LIN {X 0,Y 530.989,Z 161.345,A -85,B 0,C 180,E1 -4299.871,E2 -4299.871} C_VEL
LIN {X 0,Y 530.967,Z 161.347,A -85,B 0,C 180,E1 -4303.07,E2 -4303.07} C_VEL
LIN {X 0,Y 531.005,Z 161.342,A -85,B 0,C 180,E1 -4305.435,E2 -4305.435} C_VEL
LIN {X 0,Y 531.075,Z 161.335,A -85,B 0,C 180,E1 -4308.55,E2 -4308.55} C_VEL
LIN {X 0,Y 531.04,Z 161.335,A -85,B 0,C 180,E1 -4311.629,E2 -4311.629} C_VEL
LIN {X 0,Y 531.083,Z 161.334,A -85,B 0,C 180,E1 -4313.923,E2 -4313.923} C_VEL
LIN {X 0,Y 531.075,Z 161.333,A -85,B 0,C 180,E1 -4316.965,E2 -4316.965} C_VEL
LIN {X 0,Y 531.096,Z 161.328,A -85,B 0,C 180,E1 -4320,E2 -4320} C_VEL
LIN {X 0,Y 531.082,Z 161.331,A -85,B 0,C 180,E1 -4323.034,E2 -4323.034} C_VEL
LIN {X 0,Y 531.083,Z 161.333,A -85,B 0,C 180,E1 -4326.077,E2 -4326.077} C_VEL
LIN {X 0,Y 531.04,Z 161.334,A -85,B 0,C 180,E1 -4328.371,E2 -4328.371} C_VEL
LIN {X 0,Y 531.032,Z 161.337,A -85,B 0,C 180,E1 -4331.683,E2 -4331.683} C_VEL
LIN {X 0,Y 530.991,Z 161.345,A -85,B 0,C 180,E1 -4334.957,E2 -4334.957} C_VEL
LIN {X 0,Y 530.979,Z 161.344,A -85,B 0,C 180,E1 -4337.724,E2 -4337.724} C_VEL
LIN {X 0,Y 530.972,Z 161.343,A -85,B 0,C 180,E1 -4340.939,E2 -4340.939} C_VEL
LIN {X 0,Y 530.994,Z 161.34,A -85,B 0,C 180,E1 -4344.052,E2 -4344.052} C_VEL
LIN {X 0,Y 530.991,Z 161.344,A -85,B 0,C 180,E1 -4346.744,E2 -4346.744} C_VEL
LIN {X 0,Y 530.977,Z 161.342,A -85,B 0,C 180,E1 -4349.323,E2 -4349.323} C_VEL
LIN {X 0,Y 530.95,Z 161.35,A -85,B 0,C 180,E1 -4352.105,E2 -4352.105} C_VEL
LIN {X 0,Y 530.954,Z 161.345,A -85,B 0,C 180,E1 -4354.855,E2 -4354.855} C_VEL
LIN {X 0,Y 530.94,Z 161.351,A -85,B 0,C 180,E1 -4357.51,E2 -4357.51} C_VEL
LIN {X 0,Y 530.986,Z 161.343,A -85,B 0,C 180,E1 -4360.433,E2 -4360.433} C_VEL
LIN {X 0,Y 530.946,Z 161.345,A -85,B 0,C 180,E1 -4363.497,E2 -4363.497} C_VEL
LIN {X 0,Y 530.948,Z 161.35,A -85,B 0,C 180,E1 -4366.508,E2 -4366.508} C_VEL
LIN {X 0,Y 530.971,Z 161.346,A -85,B 0,C 180,E1 -4368.978,E2 -4368.978} C_VEL
LIN {X 0,Y 530.936,Z 161.352,A -85,B 0,C 180,E1 -4371.532,E2 -4371.532} C_VEL
LIN {X 0,Y 530.97,Z 161.357,A -85,B 0,C 180,E1 -4372.798,E2 -4372.798} C_VEL
LIN {X 0,Y 531.513,Z 165.039,A -85,B 0,C 180,E1 -4374.427,E2 -4374.427} C_VEL
LIN {X 0,Y 531.404,Z 171.668,A -85,B 0,C 180,E1 -4377.167,E2 -4377.167} C_VEL
LIN {X 0,Y 531.276,Z 179.467,A -85,B 0,C 180,E1 -4380.263,E2 -4380.263} C_VEL
LIN {X 0,Y 531.071,Z 187.303,A -85,B 0,C 180,E1 -4383.263,E2 -4383.263} C_VEL
LIN {X 0,Y 530.957,Z 194.556,A -85,B 0,C 180,E1 -4385.968,E2 -4385.968} C_VEL
LIN {X 0,Y 530.836,Z 203.007,A -85,B 0,C 180,E1 -4389.057,E2 -4389.057} C_VEL
LIN {X 0,Y 530.712,Z 211.949,A -85,B 0,C 180,E1 -4392.269,E2 -4392.269} C_VEL
LIN {X 0,Y 530.643,Z 220.324,A -85,B 0,C 180,E1 -4395.203,E2 -4395.203} C_VEL
LIN {X 0,Y 530.594,Z 223.987,A -85,B 0,C 180,E1 -4396.477,E2 -4396.477} C_VEL
LIN {X 0,Y 532.265,Z 235.706,A -85,B 0,C 180,E1 -4396.787,E2 -4396.787} C_VEL
LIN {X 0,Y 532.059,Z 248.503,A -85,B 0,C 180,E1 -4397.219,E2 -4397.219} C_VEL
LIN {X 0,Y 531.808,Z 260.711,A -85,B 0,C 180,E1 -4397.794,E2 -4397.794} C_VEL
LIN {X 0,Y 531.55,Z 271.679,A -85,B 0,C 180,E1 -4398.462,E2 -4398.462} C_VEL
LIN {X 0,Y 531.336,Z 282.994,A -85,B 0,C 180,E1 -4399.33,E2 -4399.33} C_VEL
LIN {X 0,Y 531.052,Z 292.963,A -85,B 0,C 180,E1 -4400.287,E2 -4400.287} C_VEL
LIN {X 0,Y 530.876,Z 302.631,A -85,B 0,C 180,E1 -4401.436,E2 -4401.436} C_VEL
LIN {X 0,Y 530.673,Z 310.325,A -85,B 0,C 180,E1 -4402.582,E2 -4402.582} C_VEL
LIN {X 0,Y 530.584,Z 317.42,A -85,B 0,C 180,E1 -4403.918,E2 -4403.918} C_VEL
LIN {X 0,Y 530.459,Z 322.138,A -85,B 0,C 180,E1 -4405.061,E2 -4405.061} C_VEL
LIN {X 0,Y 530.516,Z 325.746,A -85,B 0,C 180,E1 -4406.203,E2 -4406.203} C_VEL
LIN {X 0,Y 530.457,Z 327.604,A -85,B 0,C 180,E1 -4406.963,E2 -4406.963} C_VEL
LIN {X 0,Y 530.411,Z 328.997,A -85,B 0,C 180,E1 -4407.723,E2 -4407.723} C_VEL
LIN {X 0,Y 530.344,Z 330.598,A -85,B 0,C 180,E1 -4409.241,E2 -4409.241} C_VEL
LIN {X 0,Y 530.345,Z 330.814,A -85,B 0,C 180,E1 -4410.001,E2 -4410.001} C_VEL
LIN {X 0,Y 530.361,Z 329.991,A -85,B 0,C 180,E1 -4411.519,E2 -4411.519} C_VEL
LIN {X 0,Y 530.411,Z 328.998,A -85,B 0,C 180,E1 -4412.278,E2 -4412.278} C_VEL
LIN {X 0,Y 530.457,Z 327.605,A -85,B 0,C 180,E1 -4413.038,E2 -4413.038} C_VEL
LIN {X 0,Y 530.522,Z 324.673,A -85,B 0,C 180,E1 -4414.178,E2 -4414.178} C_VEL
LIN {X 0,Y 530.524,Z 320.701,A -85,B 0,C 180,E1 -4415.321,E2 -4415.321} C_VEL
LIN {X 0,Y 530.594,Z 315.01,A -85,B 0,C 180,E1 -4416.577,E2 -4416.577} C_VEL
LIN {X 0,Y 530.72,Z 307.92,A -85,B 0,C 180,E1 -4417.801,E2 -4417.801} C_VEL
LIN {X 0,Y 530.915,Z 299.639,A -85,B 0,C 180,E1 -4418.948,E2 -4418.948} C_VEL
LIN {X 0,Y 531.09,Z 291.151,A -85,B 0,C 180,E1 -4419.906,E2 -4419.906} C_VEL
LIN {X 0,Y 531.343,Z 280.664,A -85,B 0,C 180,E1 -4420.864,E2 -4420.864} C_VEL
LIN {X 0,Y 531.616,Z 268.885,A -85,B 0,C 180,E1 -4421.726,E2 -4421.726} C_VEL
LIN {X 0,Y 531.867,Z 256.995,A -85,B 0,C 180,E1 -4422.399,E2 -4422.399} C_VEL
LIN {X 0,Y 532.151,Z 244.653,A -85,B 0,C 180,E1 -4422.925,E2 -4422.925} C_VEL
LIN {X 0,Y 532.134,Z 233.818,A -85,B 0,C 180,E1 -4423.266,E2 -4423.266} C_VEL
LIN {X 0,Y 530.583,Z 223.97,A -85,B 0,C 180,E1 -4423.525,E2 -4423.525} C_VEL
LIN {X 0,Y 530.679,Z 216.462,A -85,B 0,C 180,E1 -4426.147,E2 -4426.147} C_VEL
LIN {X 0,Y 530.735,Z 208.577,A -85,B 0,C 180,E1 -4428.93,E2 -4428.93} C_VEL
LIN {X 0,Y 530.852,Z 200.724,A -85,B 0,C 180,E1 -4431.757,E2 -4431.757} C_VEL
LIN {X 0,Y 530.994,Z 192.898,A -85,B 0,C 180,E1 -4434.639,E2 -4434.639} C_VEL
LIN {X 0,Y 531.115,Z 185.096,A -85,B 0,C 180,E1 -4437.588,E2 -4437.588} C_VEL
LIN {X 0,Y 531.284,Z 178.442,A -85,B 0,C 180,E1 -4440.175,E2 -4440.175} C_VEL
LIN {X 0,Y 531.442,Z 171.845,A -85,B 0,C 180,E1 -4442.831,E2 -4442.831} C_VEL
LIN {X 0,Y 531.537,Z 165.326,A -85,B 0,C 180,E1 -4445.573,E2 -4445.573} C_VEL
LIN {X 0,Y 530.983,Z 161.348,A -85,B 0,C 180,E1 -4447.425,E2 -4447.425} C_VEL
LIN {X 0,Y 530.972,Z 161.347,A -85,B 0,C 180,E1 -4450.431,E2 -4450.431} C_VEL
LIN {X 0,Y 530.959,Z 161.347,A -85,B 0,C 180,E1 -4453.281,E2 -4453.281} C_VEL
LIN {X 0,Y 530.971,Z 161.346,A -85,B 0,C 180,E1 -4455.619,E2 -4455.619} C_VEL
LIN {X 0,Y 530.976,Z 161.346,A -85,B 0,C 180,E1 -4458.563,E2 -4458.563} C_VEL
LIN {X 0,Y 530.938,Z 161.349,A -85,B 0,C 180,E1 -4461.528,E2 -4461.528} C_VEL
LIN {X 0,Y 530.963,Z 161.343,A -85,B 0,C 180,E1 -4464.381,E2 -4464.381} C_VEL
LIN {X 0,Y 530.954,Z 161.351,A -85,B 0,C 180,E1 -4467.132,E2 -4467.132} C_VEL
LIN {X 0,Y 530.963,Z 161.345,A -85,B 0,C 180,E1 -4469.803,E2 -4469.803} C_VEL
LIN {X 0,Y 530.991,Z 161.343,A -85,B 0,C 180,E1 -4472.465,E2 -4472.465} C_VEL
LIN {X 0,Y 530.982,Z 161.343,A -85,B 0,C 180,E1 -4474.941,E2 -4474.941} C_VEL
LIN {X 0,Y 530.982,Z 161.34,A -85,B 0,C 180,E1 -4477.888,E2 -4477.888} C_VEL
LIN {X 0,Y 530.972,Z 161.347,A -85,B 0,C 180,E1 -4480.677,E2 -4480.677} C_VEL
LIN {X 0,Y 530.99,Z 161.341,A -85,B 0,C 180,E1 -4483.071,E2 -4483.071} C_VEL
LIN {X 0,Y 530.988,Z 161.345,A -85,B 0,C 180,E1 -4485.435,E2 -4485.435} C_VEL
LIN {X 0,Y 531.037,Z 161.337,A -85,B 0,C 180,E1 -4488.55,E2 -4488.55} C_VEL
LIN {X 0,Y 531.037,Z 161.334,A -85,B 0,C 180,E1 -4491.629,E2 -4491.629} C_VEL
LIN {X 0,Y 531.092,Z 161.332,A -85,B 0,C 180,E1 -4493.923,E2 -4493.923} C_VEL
LIN {X 0,Y 531.081,Z 161.333,A -85,B 0,C 180,E1 -4496.966,E2 -4496.966} C_VEL
LIN {X 0,Y 531.106,Z 161.327,A -85,B 0,C 180,E1 -4500,E2 -4500} C_VEL
LIN {X 0,Y 531.089,Z 161.328,A -85,B 0,C 180,E1 -4503.034,E2 -4503.034} C_VEL
LIN {X 0,Y 531.068,Z 161.333,A -85,B 0,C 180,E1 -4506.077,E2 -4506.077} C_VEL
LIN {X 0,Y 531.009,Z 161.343,A -85,B 0,C 180,E1 -4509.139,E2 -4509.139} C_VEL
LIN {X 0,Y 531.011,Z 161.342,A -85,B 0,C 180,E1 -4512.226,E2 -4512.226} C_VEL
LIN {X 0,Y 530.991,Z 161.342,A -85,B 0,C 180,E1 -4515.35,E2 -4515.35} C_VEL
LIN {X 0,Y 531.003,Z 161.343,A -85,B 0,C 180,E1 -4517.723,E2 -4517.723} C_VEL
LIN {X 0,Y 530.98,Z 161.347,A -85,B 0,C 180,E1 -4520.939,E2 -4520.939} C_VEL
LIN {X 0,Y 530.972,Z 161.348,A -85,B 0,C 180,E1 -4524.044,E2 -4524.044} C_VEL
LIN {X 0,Y 530.987,Z 161.341,A -85,B 0,C 180,E1 -4526.745,E2 -4526.745} C_VEL
LIN {X 0,Y 530.979,Z 161.348,A -85,B 0,C 180,E1 -4529.323,E2 -4529.323} C_VEL
LIN {X 0,Y 530.96,Z 161.345,A -85,B 0,C 180,E1 -4532.105,E2 -4532.105} C_VEL
LIN {X 0,Y 530.965,Z 161.346,A -85,B 0,C 180,E1 -4534.855,E2 -4534.855} C_VEL
LIN {X 0,Y 530.947,Z 161.351,A -85,B 0,C 180,E1 -4537.51,E2 -4537.51} C_VEL
LIN {X 0,Y 530.969,Z 161.344,A -85,B 0,C 180,E1 -4540.435,E2 -4540.435} C_VEL
LIN {X 0,Y 530.953,Z 161.346,A -85,B 0,C 180,E1 -4543.284,E2 -4543.284} C_VEL
LIN {X 0,Y 530.948,Z 161.345,A -85,B 0,C 180,E1 -4543.595,E2 -4543.595} C_VEL
LIN {X 0,Y 530.276,Z 161.434,A -85,B 0,C 180,E1 -4544.228,E2 -4544.228} C_VEL
LIN {X 0,Y 527.424,Z 161.785,A -85,B 0,C 180,E1 -4545.257,E2 -4545.257} C_VEL
LIN {X 0,Y 525.018,Z 162.089,A -85,B 0,C 180,E1 -4546.086,E2 -4546.086} C_VEL
LIN {X 0,Y 523.986,Z 162.215,A -85,B 0,C 180,E1 -4546.725,E2 -4546.725} C_VEL
LIN {X 0,Y 523.903,Z 162.224,A -85,B 0,C 180,E1 -4546.942,E2 -4546.942} C_VEL
LIN {X 0,Y 523.929,Z 162.223,A -85,B 0,C 180,E1 -4549.872,E2 -4549.872} C_VEL
LIN {X 0,Y 523.821,Z 162.236,A -85,B 0,C 180,E1 -4552.335,E2 -4552.335} C_VEL
LIN {X 0,Y 523.816,Z 162.554,A -85,B 0,C 180,E1 -4552.863,E2 -4552.863} C_VEL
LIN {X 0,Y 523.807,Z 166.831,A -85,B 0,C 180,E1 -4555.703,E2 -4555.703} C_VEL
LIN {X 0,Y 523.739,Z 171.062,A -85,B 0,C 180,E1 -4558.446,E2 -4558.446} C_VEL
LIN {X 0,Y 523.71,Z 175.251,A -85,B 0,C 180,E1 -4561.113,E2 -4561.113} C_VEL
LIN {X 0,Y 523.615,Z 180.804,A -85,B 0,C 180,E1 -4564.565,E2 -4564.565} C_VEL
LIN {X 0,Y 523.53,Z 184.955,A -85,B 0,C 180,E1 -4567.09,E2 -4567.09} C_VEL
LIN {X 0,Y 523.487,Z 190.545,A -85,B 0,C 180,E1 -4570.39,E2 -4570.39} C_VEL
LIN {X 0,Y 523.424,Z 194.766,A -85,B 0,C 180,E1 -4572.82,E2 -4572.82} C_VEL
LIN {X 0,Y 523.4,Z 197.443,A -85,B 0,C 180,E1 -4574.373,E2 -4574.373} C_VEL
LIN {X 0,Y 525.38,Z 208.957,A -85,B 0,C 180,E1 -4574.711,E2 -4574.711} C_VEL
LIN {X 0,Y 525.148,Z 221.799,A -85,B 0,C 180,E1 -4575.181,E2 -4575.181} C_VEL
LIN {X 0,Y 524.871,Z 233.415,A -85,B 0,C 180,E1 -4575.757,E2 -4575.757} C_VEL
LIN {X 0,Y 524.55,Z 244.16,A -85,B 0,C 180,E1 -4576.44,E2 -4576.44} C_VEL
LIN {X 0,Y 524.369,Z 255.094,A -85,B 0,C 180,E1 -4577.322,E2 -4577.322} C_VEL
LIN {X 0,Y 524.101,Z 264.093,A -85,B 0,C 180,E1 -4578.212,E2 -4578.212} C_VEL
LIN {X 0,Y 523.902,Z 273.617,A -85,B 0,C 180,E1 -4579.371,E2 -4579.371} C_VEL
LIN {X 0,Y 523.68,Z 281.264,A -85,B 0,C 180,E1 -4580.538,E2 -4580.538} C_VEL
LIN {X 0,Y 523.526,Z 288.298,A -85,B 0,C 180,E1 -4581.897,E2 -4581.897} C_VEL
LIN {X 0,Y 523.484,Z 292.963,A -85,B 0,C 180,E1 -4583.06,E2 -4583.06} C_VEL
LIN {X 0,Y 523.38,Z 296.521,A -85,B 0,C 180,E1 -4584.22,E2 -4584.22} C_VEL
LIN {X 0,Y 523.314,Z 299.07,A -85,B 0,C 180,E1 -4585.378,E2 -4585.378} C_VEL
LIN {X 0,Y 523.403,Z 300.265,A -85,B 0,C 180,E1 -4586.15,E2 -4586.15} C_VEL
LIN {X 0,Y 523.36,Z 301.028,A -85,B 0,C 180,E1 -4586.921,E2 -4586.921} C_VEL
LIN {X 0,Y 523.274,Z 301.383,A -85,B 0,C 180,E1 -4588.46,E2 -4588.46} C_VEL
LIN {X 0,Y 523.252,Z 300.992,A -85,B 0,C 180,E1 -4589.23,E2 -4589.23} C_VEL
LIN {X 0,Y 523.254,Z 300.182,A -85,B 0,C 180,E1 -4589.999,E2 -4589.999} C_VEL
LIN {X 0,Y 523.304,Z 297.343,A -85,B 0,C 180,E1 -4591.539,E2 -4591.539} C_VEL
LIN {X 0,Y 523.422,Z 294.095,A -85,B 0,C 180,E1 -4592.693,E2 -4592.693} C_VEL
LIN {X 0,Y 523.498,Z 289.794,A -85,B 0,C 180,E1 -4593.848,E2 -4593.848} C_VEL
LIN {X 0,Y 523.69,Z 284.313,A -85,B 0,C 180,E1 -4595.003,E2 -4595.003} C_VEL
LIN {X 0,Y 523.772,Z 277.488,A -85,B 0,C 180,E1 -4596.161,E2 -4596.161} C_VEL
LIN {X 0,Y 523.965,Z 268.939,A -85,B 0,C 180,E1 -4597.32,E2 -4597.32} C_VEL
LIN {X 0,Y 524.249,Z 260.177,A -85,B 0,C 180,E1 -4598.285,E2 -4598.285} C_VEL
LIN {X 0,Y 524.542,Z 249.398,A -85,B 0,C 180,E1 -4599.251,E2 -4599.251} C_VEL
LIN {X 0,Y 524.767,Z 238.524,A -85,B 0,C 180,E1 -4600.025,E2 -4600.025} C_VEL
LIN {X 0,Y 525.052,Z 226.348,A -85,B 0,C 180,E1 -4600.702,E2 -4600.702} C_VEL
LIN {X 0,Y 525.3,Z 214.453,A -85,B 0,C 180,E1 -4601.199,E2 -4601.199} C_VEL
LIN {X 0,Y 525.171,Z 206.737,A -85,B 0,C 180,E1 -4601.448,E2 -4601.448} C_VEL
LIN {X 0,Y 523.448,Z 197.333,A -85,B 0,C 180,E1 -4601.727,E2 -4601.727} C_VEL
LIN {X 0,Y 523.521,Z 191.992,A -85,B 0,C 180,E1 -4604.856,E2 -4604.856} C_VEL
LIN {X 0,Y 523.515,Z 186.644,A -85,B 0,C 180,E1 -4607.983,E2 -4607.983} C_VEL
LIN {X 0,Y 523.597,Z 182.589,A -85,B 0,C 180,E1 -4610.423,E2 -4610.423} C_VEL
LIN {X 0,Y 523.605,Z 178.534,A -85,B 0,C 180,E1 -4612.905,E2 -4612.905} C_VEL
LIN {X 0,Y 523.698,Z 173.624,A -85,B 0,C 180,E1 -4615.954,E2 -4615.954} C_VEL
LIN {X 0,Y 523.765,Z 169.006,A -85,B 0,C 180,E1 -4618.882,E2 -4618.882} C_VEL
LIN {X 0,Y 523.822,Z 164.876,A -85,B 0,C 180,E1 -4621.548,E2 -4621.548} C_VEL
LIN {X 0,Y 523.806,Z 162.243,A -85,B 0,C 180,E1 -4623.371,E2 -4623.371} C_VEL
LIN {X 0,Y 523.904,Z 162.228,A -85,B 0,C 180,E1 -4625.224,E2 -4625.224} C_VEL
LIN {X 0,Y 523.899,Z 162.227,A -85,B 0,C 180,E1 -4628.099,E2 -4628.099} C_VEL
LIN {X 0,Y 523.946,Z 162.219,A -85,B 0,C 180,E1 -4631.308,E2 -4631.308} C_VEL
LIN {X 0,Y 523.938,Z 162.219,A -85,B 0,C 180,E1 -4634.689,E2 -4634.689} C_VEL
LIN {X 0,Y 523.946,Z 162.217,A -85,B 0,C 180,E1 -4637.88,E2 -4637.88} C_VEL
LIN {X 0,Y 523.908,Z 162.227,A -85,B 0,C 180,E1 -4640.914,E2 -4640.914} C_VEL
LIN {X 0,Y 523.879,Z 162.229,A -85,B 0,C 180,E1 -4643.823,E2 -4643.823} C_VEL
LIN {X 0,Y 523.916,Z 162.223,A -85,B 0,C 180,E1 -4646.633,E2 -4646.633} C_VEL
LIN {X 0,Y 523.935,Z 162.224,A -85,B 0,C 180,E1 -4649.354,E2 -4649.354} C_VEL
LIN {X 0,Y 523.953,Z 162.217,A -85,B 0,C 180,E1 -4652.278,E2 -4652.278} C_VEL
LIN {X 0,Y 523.954,Z 162.223,A -85,B 0,C 180,E1 -4654.581,E2 -4654.581} C_VEL
LIN {X 0,Y 523.932,Z 162.219,A -85,B 0,C 180,E1 -4657.107,E2 -4657.107} C_VEL
LIN {X 0,Y 523.943,Z 162.223,A -85,B 0,C 180,E1 -4659.864,E2 -4659.864} C_VEL
LIN {X 0,Y 523.941,Z 162.22,A -85,B 0,C 180,E1 -4662.836,E2 -4662.836} C_VEL
LIN {X 0,Y 523.968,Z 162.219,A -85,B 0,C 180,E1 -4665.235,E2 -4665.235} C_VEL
LIN {X 0,Y 524.029,Z 162.212,A -85,B 0,C 180,E1 -4668.394,E2 -4668.394} C_VEL
LIN {X 0,Y 523.985,Z 162.213,A -85,B 0,C 180,E1 -4671.515,E2 -4671.515} C_VEL
LIN {X 0,Y 524.041,Z 162.212,A -85,B 0,C 180,E1 -4673.841,E2 -4673.841} C_VEL
LIN {X 0,Y 524.041,Z 162.208,A -85,B 0,C 180,E1 -4676.925,E2 -4676.925} C_VEL
LIN {X 0,Y 524.068,Z 162.203,A -85,B 0,C 180,E1 -4680,E2 -4680} C_VEL
LIN {X 0,Y 524.048,Z 162.207,A -85,B 0,C 180,E1 -4683.075,E2 -4683.075} C_VEL
LIN {X 0,Y 524.039,Z 162.21,A -85,B 0,C 180,E1 -4686.159,E2 -4686.159} C_VEL
LIN {X 0,Y 523.984,Z 162.212,A -85,B 0,C 180,E1 -4688.484,E2 -4688.484} C_VEL
LIN {X 0,Y 524.005,Z 162.211,A -85,B 0,C 180,E1 -4691.762,E2 -4691.762} C_VEL
LIN {X 0,Y 523.955,Z 162.22,A -85,B 0,C 180,E1 -4695.054,E2 -4695.054} C_VEL
LIN {X 0,Y 523.927,Z 162.225,A -85,B 0,C 180,E1 -4697.97,E2 -4697.97} C_VEL
LIN {X 0,Y 523.938,Z 162.221,A -85,B 0,C 180,E1 -4700.411,E2 -4700.411} C_VEL
LIN {X 0,Y 523.931,Z 162.221,A -85,B 0,C 180,E1 -4702.893,E2 -4702.893} C_VEL
LIN {X 0,Y 523.953,Z 162.22,A -85,B 0,C 180,E1 -4705.419,E2 -4705.419} C_VEL
LIN {X 0,Y 523.942,Z 162.217,A -85,B 0,C 180,E1 -4708,E2 -4708} C_VEL
LIN {X 0,Y 523.922,Z 162.223,A -85,B 0,C 180,E1 -4710.858,E2 -4710.858} C_VEL
LIN {X 0,Y 523.931,Z 162.224,A -85,B 0,C 180,E1 -4713.737,E2 -4713.737} C_VEL
LIN {X 0,Y 523.893,Z 162.225,A -85,B 0,C 180,E1 -4716.406,E2 -4716.406} C_VEL
LIN {X 0,Y 523.935,Z 162.224,A -85,B 0,C 180,E1 -4719.084,E2 -4719.084} C_VEL
LIN {X 0,Y 523.944,Z 162.219,A -85,B 0,C 180,E1 -4722.12,E2 -4722.12} C_VEL
LIN {X 0,Y 523.935,Z 162.218,A -85,B 0,C 180,E1 -4725.311,E2 -4725.311} C_VEL
LIN {X 0,Y 523.944,Z 162.221,A -85,B 0,C 180,E1 -4728.691,E2 -4728.691} C_VEL
LIN {X 0,Y 523.897,Z 162.229,A -85,B 0,C 180,E1 -4731.901,E2 -4731.901} C_VEL
LIN {X 0,Y 523.93,Z 162.314,A -85,B 0,C 180,E1 -4732.67,E2 -4732.67} C_VEL
LIN {X 0,Y 524.535,Z 167.151,A -85,B 0,C 180,E1 -4734.824,E2 -4734.824} C_VEL
LIN {X 0,Y 524.353,Z 173.853,A -85,B 0,C 180,E1 -4737.608,E2 -4737.608} C_VEL
LIN {X 0,Y 524.232,Z 181.379,A -85,B 0,C 180,E1 -4740.623,E2 -4740.623} C_VEL
LIN {X 0,Y 524.004,Z 190.068,A -85,B 0,C 180,E1 -4743.976,E2 -4743.976} C_VEL
LIN {X 0,Y 523.838,Z 197.286,A -85,B 0,C 180,E1 -4746.688,E2 -4746.688} C_VEL
LIN {X 0,Y 523.717,Z 205.117,A -85,B 0,C 180,E1 -4749.582,E2 -4749.582} C_VEL
LIN {X 0,Y 523.614,Z 212.762,A -85,B 0,C 180,E1 -4752.359,E2 -4752.359} C_VEL
LIN {X 0,Y 523.565,Z 220.777,A -85,B 0,C 180,E1 -4755.225,E2 -4755.225} C_VEL
LIN {X 0,Y 523.541,Z 223.785,A -85,B 0,C 180,E1 -4756.291,E2 -4756.291} C_VEL
LIN {X 0,Y 525.347,Z 236.422,A -85,B 0,C 180,E1 -4756.635,E2 -4756.635} C_VEL
LIN {X 0,Y 525.092,Z 249.437,A -85,B 0,C 180,E1 -4757.096,E2 -4757.096} C_VEL
LIN {X 0,Y 524.803,Z 261.775,A -85,B 0,C 180,E1 -4757.699,E2 -4757.699} C_VEL
LIN {X 0,Y 524.553,Z 272.96,A -85,B 0,C 180,E1 -4758.408,E2 -4758.408} C_VEL
LIN {X 0,Y 524.288,Z 283.868,A -85,B 0,C 180,E1 -4759.282,E2 -4759.282} C_VEL
LIN {X 0,Y 524.025,Z 292.765,A -85,B 0,C 180,E1 -4760.155,E2 -4760.155} C_VEL
LIN {X 0,Y 523.809,Z 302.433,A -85,B 0,C 180,E1 -4761.32,E2 -4761.32} C_VEL
LIN {X 0,Y 523.602,Z 310.127,A -85,B 0,C 180,E1 -4762.481,E2 -4762.481} C_VEL
LIN {X 0,Y 523.479,Z 317.222,A -85,B 0,C 180,E1 -4763.835,E2 -4763.835} C_VEL
LIN {X 0,Y 523.383,Z 321.94,A -85,B 0,C 180,E1 -4764.994,E2 -4764.994} C_VEL
LIN {X 0,Y 523.443,Z 325.548,A -85,B 0,C 180,E1 -4766.152,E2 -4766.152} C_VEL
LIN {X 0,Y 523.367,Z 327.406,A -85,B 0,C 180,E1 -4766.922,E2 -4766.922} C_VEL
LIN {X 0,Y 523.335,Z 328.8,A -85,B 0,C 180,E1 -4767.692,E2 -4767.692} C_VEL
LIN {X 0,Y 523.25,Z 330.4,A -85,B 0,C 180,E1 -4769.231,E2 -4769.231} C_VEL
LIN {X 0,Y 523.249,Z 330.616,A -85,B 0,C 180,E1 -4770.001,E2 -4770.001} C_VEL
LIN {X 0,Y 523.274,Z 329.794,A -85,B 0,C 180,E1 -4771.54,E2 -4771.54} C_VEL
LIN {X 0,Y 523.335,Z 328.801,A -85,B 0,C 180,E1 -4772.309,E2 -4772.309} C_VEL
LIN {X 0,Y 523.367,Z 327.407,A -85,B 0,C 180,E1 -4773.079,E2 -4773.079} C_VEL
LIN {X 0,Y 523.424,Z 324.474,A -85,B 0,C 180,E1 -4774.235,E2 -4774.235} C_VEL
LIN {X 0,Y 523.461,Z 320.503,A -85,B 0,C 180,E1 -4775.393,E2 -4775.393} C_VEL
LIN {X 0,Y 523.514,Z 315.296,A -85,B 0,C 180,E1 -4776.572,E2 -4776.572} C_VEL
LIN {X 0,Y 523.639,Z 308.958,A -85,B 0,C 180,E1 -4777.713,E2 -4777.713} C_VEL
LIN {X 0,Y 523.823,Z 300.931,A -85,B 0,C 180,E1 -4778.876,E2 -4778.876} C_VEL
LIN {X 0,Y 524.026,Z 292.751,A -85,B 0,C 180,E1 -4779.846,E2 -4779.846} C_VEL
LIN {X 0,Y 524.308,Z 282.779,A -85,B 0,C 180,E1 -4780.816,E2 -4780.816} C_VEL
LIN {X 0,Y 524.573,Z 271.603,A -85,B 0,C 180,E1 -4781.685,E2 -4781.685} C_VEL
LIN {X 0,Y 524.826,Z 260.488,A -85,B 0,C 180,E1 -4782.372,E2 -4782.372} C_VEL
LIN {X 0,Y 525.135,Z 248.267,A -85,B 0,C 180,E1 -4782.954,E2 -4782.954} C_VEL
LIN {X 0,Y 525.299,Z 235.224,A -85,B 0,C 180,E1 -4783.398,E2 -4783.398} C_VEL
LIN {X 0,Y 523.528,Z 223.768,A -85,B 0,C 180,E1 -4783.71,E2 -4783.71} C_VEL
LIN {X 0,Y 523.611,Z 215.13,A -85,B 0,C 180,E1 -4786.772,E2 -4786.772} C_VEL
LIN {X 0,Y 523.715,Z 207.341,A -85,B 0,C 180,E1 -4789.601,E2 -4789.601} C_VEL
LIN {X 0,Y 523.806,Z 200.223,A -85,B 0,C 180,E1 -4792.212,E2 -4792.212} C_VEL
LIN {X 0,Y 523.95,Z 192.799,A -85,B 0,C 180,E1 -4794.993,E2 -4794.993} C_VEL
LIN {X 0,Y 524.143,Z 185.021,A -85,B 0,C 180,E1 -4797.987,E2 -4797.987} C_VEL
LIN {X 0,Y 524.298,Z 177.65,A -85,B 0,C 180,E1 -4800.919,E2 -4800.919} C_VEL
LIN {X 0,Y 524.468,Z 170.64,A -85,B 0,C 180,E1 -4803.817,E2 -4803.817} C_VEL
LIN {X 0,Y 524.535,Z 166.383,A -85,B 0,C 180,E1 -4805.647,E2 -4805.647} C_VEL
LIN {X 0,Y 523.942,Z 162.224,A -85,B 0,C 180,E1 -4807.614,E2 -4807.614} C_VEL
LIN {X 0,Y 523.926,Z 162.228,A -85,B 0,C 180,E1 -4810.128,E2 -4810.128} C_VEL
LIN {X 0,Y 523.928,Z 162.221,A -85,B 0,C 180,E1 -4812.458,E2 -4812.458} C_VEL
LIN {X 0,Y 523.94,Z 162.224,A -85,B 0,C 180,E1 -4815.307,E2 -4815.307} C_VEL
LIN {X 0,Y 523.939,Z 162.223,A -85,B 0,C 180,E1 -4818.688,E2 -4818.688} C_VEL
LIN {X 0,Y 523.899,Z 162.225,A -85,B 0,C 180,E1 -4821.079,E2 -4821.079} C_VEL
LIN {X 0,Y 523.91,Z 162.226,A -85,B 0,C 180,E1 -4823.826,E2 -4823.826} C_VEL
LIN {X 0,Y 523.923,Z 162.222,A -85,B 0,C 180,E1 -4826.634,E2 -4826.634} C_VEL
LIN {X 0,Y 523.941,Z 162.22,A -85,B 0,C 180,E1 -4829.355,E2 -4829.355} C_VEL
LIN {X 0,Y 523.954,Z 162.221,A -85,B 0,C 180,E1 -4832.28,E2 -4832.28} C_VEL
LIN {X 0,Y 523.928,Z 162.221,A -85,B 0,C 180,E1 -4834.58,E2 -4834.58} C_VEL
LIN {X 0,Y 523.935,Z 162.225,A -85,B 0,C 180,E1 -4837.108,E2 -4837.108} C_VEL
LIN {X 0,Y 523.952,Z 162.217,A -85,B 0,C 180,E1 -4839.865,E2 -4839.865} C_VEL
LIN {X 0,Y 523.969,Z 162.216,A -85,B 0,C 180,E1 -4842.837,E2 -4842.837} C_VEL
LIN {X 0,Y 523.946,Z 162.222,A -85,B 0,C 180,E1 -4845.235,E2 -4845.235} C_VEL
LIN {X 0,Y 524.01,Z 162.211,A -85,B 0,C 180,E1 -4848.394,E2 -4848.394} C_VEL
LIN {X 0,Y 523.985,Z 162.212,A -85,B 0,C 180,E1 -4851.516,E2 -4851.516} C_VEL
LIN {X 0,Y 524.05,Z 162.209,A -85,B 0,C 180,E1 -4853.841,E2 -4853.841} C_VEL
LIN {X 0,Y 524.047,Z 162.208,A -85,B 0,C 180,E1 -4856.925,E2 -4856.925} C_VEL
LIN {X 0,Y 524.077,Z 162.203,A -85,B 0,C 180,E1 -4860,E2 -4860} C_VEL
LIN {X 0,Y 524.055,Z 162.204,A -85,B 0,C 180,E1 -4863.075,E2 -4863.075} C_VEL
LIN {X 0,Y 524.028,Z 162.21,A -85,B 0,C 180,E1 -4866.159,E2 -4866.159} C_VEL
LIN {X 0,Y 523.977,Z 162.219,A -85,B 0,C 180,E1 -4869.262,E2 -4869.262} C_VEL
LIN {X 0,Y 523.975,Z 162.216,A -85,B 0,C 180,E1 -4871.741,E2 -4871.741} C_VEL
LIN {X 0,Y 523.963,Z 162.216,A -85,B 0,C 180,E1 -4875.053,E2 -4875.053} C_VEL
LIN {X 0,Y 523.946,Z 162.219,A -85,B 0,C 180,E1 -4877.97,E2 -4877.97} C_VEL
LIN {X 0,Y 523.948,Z 162.22,A -85,B 0,C 180,E1 -4880.411,E2 -4880.411} C_VEL
LIN {X 0,Y 523.907,Z 162.226,A -85,B 0,C 180,E1 -4882.894,E2 -4882.894} C_VEL
LIN {X 0,Y 523.962,Z 162.22,A -85,B 0,C 180,E1 -4886.022,E2 -4886.022} C_VEL
LIN {X 0,Y 523.929,Z 162.221,A -85,B 0,C 180,E1 -4888.876,E2 -4888.876} C_VEL
LIN {X 0,Y 523.912,Z 162.223,A -85,B 0,C 180,E1 -4891.545,E2 -4891.545} C_VEL
LIN {X 0,Y 523.923,Z 162.225,A -85,B 0,C 180,E1 -4894.291,E2 -4894.291} C_VEL
LIN {X 0,Y 523.892,Z 162.227,A -85,B 0,C 180,E1 -4897.134,E2 -4897.134} C_VEL
LIN {X 0,Y 523.922,Z 162.221,A -85,B 0,C 180,E1 -4900.132,E2 -4900.132} C_VEL
LIN {X 0,Y 523.924,Z 162.223,A -85,B 0,C 180,E1 -4902.461,E2 -4902.461} C_VEL
LIN {X 0,Y 523.942,Z 162.219,A -85,B 0,C 180,E1 -4905.311,E2 -4905.311} C_VEL
LIN {X 0,Y 523.903,Z 162.224,A -85,B 0,C 180,E1 -4906.942,E2 -4906.942} C_VEL
LIN {X 0,Y 523.237,Z 162.31,A -85,B 0,C 180,E1 -4907.584,E2 -4907.584} C_VEL
LIN {X 0,Y 520.381,Z 162.663,A -85,B 0,C 180,E1 -4908.625,E2 -4908.625} C_VEL
LIN {X 0,Y 517.968,Z 162.966,A -85,B 0,C 180,E1 -4909.464,E2 -4909.464} C_VEL
LIN {X 0,Y 516.934,Z 163.093,A -85,B 0,C 180,E1 -4910.112,E2 -4910.112} C_VEL
LIN {X 0,Y 516.851,Z 163.103,A -85,B 0,C 180,E1 -4910.332,E2 -4910.332} C_VEL
LIN {X 0,Y 516.782,Z 163.113,A -85,B 0,C 180,E1 -4912.27,E2 -4912.27} C_VEL
LIN {X 0,Y 516.769,Z 164.191,A -85,B 0,C 180,E1 -4913.36,E2 -4913.36} C_VEL
LIN {X 0,Y 516.753,Z 168.287,A -85,B 0,C 180,E1 -4916.111,E2 -4916.111} C_VEL
LIN {X 0,Y 516.669,Z 172.678,A -85,B 0,C 180,E1 -4918.978,E2 -4918.978} C_VEL
LIN {X 0,Y 516.615,Z 176.715,A -85,B 0,C 180,E1 -4921.568,E2 -4921.568} C_VEL
LIN {X 0,Y 516.545,Z 182.272,A -85,B 0,C 180,E1 -4925.054,E2 -4925.054} C_VEL
LIN {X 0,Y 516.426,Z 186.634,A -85,B 0,C 180,E1 -4927.731,E2 -4927.731} C_VEL
